LIN {X 0,Y 573.962,Z 477.903,A -85,B 0,C 180,E1 -2264.781,E2 -2264.781} C_VEL
LIN {X 0,Y 574.142,Z 465.512,A -85,B 0,C 180,E1 -2265.532,E2 -2265.532} C_VEL
LIN {X 0,Y 574.337,Z 450.828,A -85,B 0,C 180,E1 -2266.255,E2 -2266.255} C_VEL
LIN {X 0,Y 574.546,Z 436.614,A -85,B 0,C 180,E1 -2266.797,E2 -2266.797} C_VEL
LIN {X 0,Y 574.665,Z 421.538,A -85,B 0,C 180,E1 -2267.224,E2 -2267.224} C_VEL
LIN {X 0,Y 574.759,Z 406.593,A -85,B 0,C 180,E1 -2267.503,E2 -2267.503} C_VEL
LIN {X 0,Y 575.2,Z 251.055,A -85,B 0,C 180,E1 -2269.501,E2 -2269.501} C_VEL
LIN {X 0,Y 574.168,Z 244.937,A -85,B 0,C 180,E1 -2269.638,E2 -2269.638} C_VEL
LIN {X 0,Y 574.518,Z 217.413,A -85,B 0,C 180,E1 -2272.475,E2 -2272.475} C_VEL
LIN {X 0,Y 574.959,Z 188.463,A -85,B 0,C 180,E1 -2275.523,E2 -2275.523} C_VEL
LIN {X 0,Y 573.783,Z 183.004,A -85,B 0,C 180,E1 -2276.164,E2 -2276.164} C_VEL
LIN {X 0,Y 573.246,Z 180.78,A -85,B 0,C 180,E1 -2276.472,E2 -2276.472} C_VEL
LIN {X 0,Y 573.227,Z 180.7,A -85,B 0,C 180,E1 -2278.565,E2 -2278.565} C_VEL
LIN {X 0,Y 573.216,Z 180.692,A -85,B 0,C 180,E1 -2280.994,E2 -2280.994} C_VEL
LIN {X 0,Y 573.24,Z 180.703,A -85,B 0,C 180,E1 -2283.521,E2 -2283.521} C_VEL
LIN {X 0,Y 573.212,Z 180.701,A -85,B 0,C 180,E1 -2286.051,E2 -2286.051} C_VEL
LIN {X 0,Y 573.235,Z 180.708,A -85,B 0,C 180,E1 -2288.702,E2 -2288.702} C_VEL
LIN {X 0,Y 573.224,Z 180.702,A -85,B 0,C 180,E1 -2291.592,E2 -2291.592} C_VEL
LIN {X 0,Y 573.22,Z 180.705,A -85,B 0,C 180,E1 -2294.335,E2 -2294.335} C_VEL
LIN {X 0,Y 573.237,Z 180.699,A -85,B 0,C 180,E1 -2297.358,E2 -2297.358} C_VEL
LIN {X 0,Y 573.242,Z 180.706,A -85,B 0,C 180,E1 -2300.393,E2 -2300.393} C_VEL
LIN {X 0,Y 573.249,Z 180.7,A -85,B 0,C 180,E1 -2303.077,E2 -2303.077} C_VEL
LIN {X 0,Y 573.264,Z 180.697,A -85,B 0,C 180,E1 -2305.671,E2 -2305.671} C_VEL
LIN {X 0,Y 573.242,Z 180.702,A -85,B 0,C 180,E1 -2308.185,E2 -2308.185} C_VEL
LIN {X 0,Y 573.256,Z 180.702,A -85,B 0,C 180,E1 -2310.634,E2 -2310.634} C_VEL
LIN {X 0,Y 573.248,Z 180.695,A -85,B 0,C 180,E1 -2313.024,E2 -2313.024} C_VEL
LIN {X 0,Y 573.272,Z 180.695,A -85,B 0,C 180,E1 -2315.366,E2 -2315.366} C_VEL
LIN {X 0,Y 573.223,Z 180.707,A -85,B 0,C 180,E1 -2318.419,E2 -2318.419} C_VEL
LIN {X 0,Y 573.265,Z 180.697,A -85,B 0,C 180,E1 -2320.731,E2 -2320.731} C_VEL
LIN {X 0,Y 573.24,Z 180.703,A -85,B 0,C 180,E1 -2323.622,E2 -2323.622} C_VEL
LIN {X 0,Y 573.271,Z 180.702,A -85,B 0,C 180,E1 -2325.807,E2 -2325.807} C_VEL
LIN {X 0,Y 573.259,Z 180.697,A -85,B 0,C 180,E1 -2328.745,E2 -2328.745} C_VEL
LIN {X 0,Y 573.28,Z 180.699,A -85,B 0,C 180,E1 -2331.541,E2 -2331.541} C_VEL
LIN {X 0,Y 573.288,Z 180.694,A -85,B 0,C 180,E1 -2334.372,E2 -2334.372} C_VEL
LIN {X 0,Y 573.305,Z 180.696,A -85,B 0,C 180,E1 -2337.893,E2 -2337.893} C_VEL
LIN {X 0,Y 573.329,Z 180.688,A -85,B 0,C 180,E1 -2340.702,E2 -2340.702} C_VEL
LIN {X 0,Y 573.232,Z 180.708,A -85,B 0,C 180,E1 -2343.515,E2 -2343.515} C_VEL
LIN {X 0,Y 573.287,Z 180.701,A -85,B 0,C 180,E1 -2345.628,E2 -2345.628} C_VEL
LIN {X 0,Y 573.287,Z 180.693,A -85,B 0,C 180,E1 -2348.46,E2 -2348.46} C_VEL
LIN {X 0,Y 573.269,Z 180.705,A -85,B 0,C 180,E1 -2351.312,E2 -2351.312} C_VEL
LIN {X 0,Y 573.271,Z 180.696,A -85,B 0,C 180,E1 -2354.193,E2 -2354.193} C_VEL
LIN {X 0,Y 573.256,Z 180.704,A -85,B 0,C 180,E1 -2357.112,E2 -2357.112} C_VEL
LIN {X 0,Y 573.25,Z 180.697,A -85,B 0,C 180,E1 -2360.077,E2 -2360.077} C_VEL
LIN {X 0,Y 573.232,Z 180.709,A -85,B 0,C 180,E1 -2363.1,E2 -2363.1} C_VEL
LIN {X 0,Y 573.248,Z 180.699,A -85,B 0,C 180,E1 -2364.391,E2 -2364.391} C_VEL
LIN {X 0,Y 572.622,Z 180.785,A -85,B 0,C 180,E1 -2364.977,E2 -2364.977} C_VEL
LIN {X 0,Y 569.78,Z 181.138,A -85,B 0,C 180,E1 -2365.928,E2 -2365.928} C_VEL
LIN {X 0,Y 567.347,Z 181.439,A -85,B 0,C 180,E1 -2366.694,E2 -2366.694} C_VEL
LIN {X 0,Y 566.291,Z 181.568,A -85,B 0,C 180,E1 -2367.285,E2 -2367.285} C_VEL
LIN {X 0,Y 566.201,Z 181.576,A -85,B 0,C 180,E1 -2367.485,E2 -2367.485} C_VEL
LIN {X 0,Y 566.2,Z 181.575,A -85,B 0,C 180,E1 -2369.769,E2 -2369.769} C_VEL
LIN {X 0,Y 566.201,Z 181.58,A -85,B 0,C 180,E1 -2372.43,E2 -2372.43} C_VEL
LIN {X 0,Y 566.213,Z 181.58,A -85,B 0,C 180,E1 -2374.995,E2 -2374.995} C_VEL
LIN {X 0,Y 566.196,Z 181.578,A -85,B 0,C 180,E1 -2377.461,E2 -2377.461} C_VEL
LIN {X 0,Y 566.206,Z 181.576,A -85,B 0,C 180,E1 -2380.199,E2 -2380.199} C_VEL
LIN {X 0,Y 566.199,Z 181.578,A -85,B 0,C 180,E1 -2383.055,E2 -2383.055} C_VEL
LIN {X 0,Y 566.198,Z 181.58,A -85,B 0,C 180,E1 -2386.049,E2 -2386.049} C_VEL
LIN {X 0,Y 566.182,Z 181.583,A -85,B 0,C 180,E1 -2388.861,E2 -2388.861} C_VEL
LIN {X 0,Y 566.183,Z 181.579,A -85,B 0,C 180,E1 -2391.637,E2 -2391.637} C_VEL
LIN {X 0,Y 566.192,Z 181.586,A -85,B 0,C 180,E1 -2394.31,E2 -2394.31} C_VEL
LIN {X 0,Y 566.221,Z 181.573,A -85,B 0,C 180,E1 -2396.898,E2 -2396.898} C_VEL
LIN {X 0,Y 566.18,Z 181.58,A -85,B 0,C 180,E1 -2399.407,E2 -2399.407} C_VEL
LIN {X 0,Y 566.189,Z 181.586,A -85,B 0,C 180,E1 -2401.856,E2 -2401.856} C_VEL
LIN {X 0,Y 566.246,Z 181.778,A -85,B 0,C 180,E1 -2404.742,E2 -2404.742} C_VEL
LIN {X 0,Y 567.586,Z 188.138,A -85,B 0,C 180,E1 -2405.688,E2 -2405.688} C_VEL
LIN {X 0,Y 567.264,Z 206.844,A -85,B 0,C 180,E1 -2408.181,E2 -2408.181} C_VEL
LIN {X 0,Y 566.942,Z 228.424,A -85,B 0,C 180,E1 -2411.01,E2 -2411.01} C_VEL
LIN {X 0,Y 566.745,Z 244.508,A -85,B 0,C 180,E1 -2413.048,E2 -2413.048} C_VEL
LIN {X 0,Y 567.822,Z 250.993,A -85,B 0,C 180,E1 -2413.189,E2 -2413.189} C_VEL
LIN {X 0,Y 567.418,Z 382.93,A -85,B 0,C 180,E1 -2414.901,E2 -2414.901} C_VEL
LIN {X 0,Y 567.322,Z 397.304,A -85,B 0,C 180,E1 -2415.239,E2 -2415.239} C_VEL
LIN {X 0,Y 567.132,Z 411.854,A -85,B 0,C 180,E1 -2415.742,E2 -2415.742} C_VEL
LIN {X 0,Y 566.944,Z 425.536,A -85,B 0,C 180,E1 -2416.377,E2 -2416.377} C_VEL
LIN {X 0,Y 566.745,Z 437.822,A -85,B 0,C 180,E1 -2417.102,E2 -2417.102} C_VEL
LIN {X 0,Y 566.56,Z 450.215,A -85,B 0,C 180,E1 -2418.008,E2 -2418.008} C_VEL
LIN {X 0,Y 566.435,Z 461.051,A -85,B 0,C 180,E1 -2418.979,E2 -2418.979} C_VEL
LIN {X 0,Y 566.215,Z 470.48,A -85,B 0,C 180,E1 -2419.993,E2 -2419.993} C_VEL
LIN {X 0,Y 566.133,Z 478.863,A -85,B 0,C 180,E1 -2421.073,E2 -2421.073} C_VEL
LIN {X 0,Y 566.047,Z 486.874,A -85,B 0,C 180,E1 -2422.33,E2 -2422.33} C_VEL
LIN {X 0,Y 565.945,Z 493.325,A -85,B 0,C 180,E1 -2423.583,E2 -2423.583} C_VEL
LIN {X 0,Y 565.928,Z 497.799,A -85,B 0,C 180,E1 -2424.656,E2 -2424.656} C_VEL
LIN {X 0,Y 565.957,Z 501.312,A -85,B 0,C 180,E1 -2425.727,E2 -2425.727} C_VEL
LIN {X 0,Y 565.875,Z 504.745,A -85,B 0,C 180,E1 -2427.152,E2 -2427.152} C_VEL
LIN {X 0,Y 565.844,Z 506.786,A -85,B 0,C 180,E1 -2428.576,E2 -2428.576} C_VEL
LIN {X 0,Y 565.838,Z 507.496,A -85,B 0,C 180,E1 -2430,E2 -2430} C_VEL
LIN {X 0,Y 565.841,Z 506.882,A -85,B 0,C 180,E1 -2431.423,E2 -2431.423} C_VEL
LIN {X 0,Y 565.873,Z 504.926,A -85,B 0,C 180,E1 -2432.847,E2 -2432.847} C_VEL
LIN {X 0,Y 565.958,Z 501.581,A -85,B 0,C 180,E1 -2434.273,E2 -2434.273} C_VEL
LIN {X 0,Y 565.983,Z 496.748,A -85,B 0,C 180,E1 -2435.701,E2 -2435.701} C_VEL
LIN {X 0,Y 565.98,Z 490.283,A -85,B 0,C 180,E1 -2437.133,E2 -2437.133} C_VEL
LIN {X 0,Y 566.093,Z 483.082,A -85,B 0,C 180,E1 -2438.388,E2 -2438.388} C_VEL
LIN {X 0,Y 566.172,Z 475.542,A -85,B 0,C 180,E1 -2439.466,E2 -2439.466} C_VEL
LIN {X 0,Y 566.29,Z 466.488,A -85,B 0,C 180,E1 -2440.547,E2 -2440.547} C_VEL
LIN {X 0,Y 566.47,Z 455.522,A -85,B 0,C 180,E1 -2441.631,E2 -2441.631} C_VEL
LIN {X 0,Y 566.642,Z 444.356,A -85,B 0,C 180,E1 -2442.535,E2 -2442.535} C_VEL
LIN {X 0,Y 566.843,Z 432.011,A -85,B 0,C 180,E1 -2443.351,E2 -2443.351} C_VEL
LIN {X 0,Y 567.065,Z 420.127,A -85,B 0,C 180,E1 -2443.985,E2 -2443.985} C_VEL
LIN {X 0,Y 567.232,Z 407.918,A -85,B 0,C 180,E1 -2444.503,E2 -2444.503} C_VEL
LIN {X 0,Y 567.343,Z 393.992,A -85,B 0,C 180,E1 -2444.943,E2 -2444.943} C_VEL
LIN {X 0,Y 567.428,Z 380.103,A -85,B 0,C 180,E1 -2445.236,E2 -2445.236} C_VEL
LIN {X 0,Y 567.751,Z 250.574,A -85,B 0,C 180,E1 -2446.908,E2 -2446.908} C_VEL
LIN {X 0,Y 566.728,Z 244.432,A -85,B 0,C 180,E1 -2447.047,E2 -2447.047} C_VEL
LIN {X 0,Y 566.979,Z 224.441,A -85,B 0,C 180,E1 -2449.599,E2 -2449.599} C_VEL
LIN {X 0,Y 567.381,Z 201.774,A -85,B 0,C 180,E1 -2452.58,E2 -2452.58} C_VEL
LIN {X 0,Y 567.58,Z 188.81,A -85,B 0,C 180,E1 -2454.312,E2 -2454.312} C_VEL
LIN {X 0,Y 566.223,Z 181.721,A -85,B 0,C 180,E1 -2455.363,E2 -2455.363} C_VEL
LIN {X 0,Y 566.184,Z 181.587,A -85,B 0,C 180,E1 -2458.198,E2 -2458.198} C_VEL
LIN {X 0,Y 566.188,Z 181.579,A -85,B 0,C 180,E1 -2461.075,E2 -2461.075} C_VEL
LIN {X 0,Y 566.21,Z 181.578,A -85,B 0,C 180,E1 -2463.733,E2 -2463.733} C_VEL
LIN {X 0,Y 566.212,Z 181.575,A -85,B 0,C 180,E1 -2466.568,E2 -2466.568} C_VEL
LIN {X 0,Y 566.212,Z 181.583,A -85,B 0,C 180,E1 -2469.685,E2 -2469.685} C_VEL
LIN {X 0,Y 566.21,Z 181.577,A -85,B 0,C 180,E1 -2472.087,E2 -2472.087} C_VEL
LIN {X 0,Y 566.17,Z 181.583,A -85,B 0,C 180,E1 -2475.035,E2 -2475.035} C_VEL
LIN {X 0,Y 566.214,Z 181.576,A -85,B 0,C 180,E1 -2478.135,E2 -2478.135} C_VEL
LIN {X 0,Y 566.211,Z 181.574,A -85,B 0,C 180,E1 -2480.726,E2 -2480.726} C_VEL
LIN {X 0,Y 566.213,Z 181.577,A -85,B 0,C 180,E1 -2483.783,E2 -2483.783} C_VEL
LIN {X 0,Y 566.207,Z 181.574,A -85,B 0,C 180,E1 -2486.265,E2 -2486.265} C_VEL
LIN {X 0,Y 566.193,Z 181.583,A -85,B 0,C 180,E1 -2488.922,E2 -2488.922} C_VEL
LIN {X 0,Y 566.19,Z 181.582,A -85,B 0,C 180,E1 -2491.046,E2 -2491.046} C_VEL
LIN {X 0,Y 566.21,Z 181.579,A -85,B 0,C 180,E1 -2493.458,E2 -2493.458} C_VEL
LIN {X 0,Y 566.193,Z 181.577,A -85,B 0,C 180,E1 -2495.819,E2 -2495.819} C_VEL
LIN {X 0,Y 566.202,Z 181.586,A -85,B 0,C 180,E1 -2498.902,E2 -2498.902} C_VEL
LIN {X 0,Y 566.206,Z 181.581,A -85,B 0,C 180,E1 -2501.172,E2 -2501.172} C_VEL
LIN {X 0,Y 566.215,Z 181.575,A -85,B 0,C 180,E1 -2503.412,E2 -2503.412} C_VEL
LIN {X 0,Y 566.195,Z 181.581,A -85,B 0,C 180,E1 -2506.359,E2 -2506.359} C_VEL
LIN {X 0,Y 566.227,Z 181.581,A -85,B 0,C 180,E1 -2508.675,E2 -2508.675} C_VEL
LIN {X 0,Y 566.227,Z 181.573,A -85,B 0,C 180,E1 -2511.434,E2 -2511.434} C_VEL
LIN {X 0,Y 566.254,Z 181.575,A -85,B 0,C 180,E1 -2514.302,E2 -2514.302} C_VEL
LIN {X 0,Y 566.274,Z 181.568,A -85,B 0,C 180,E1 -2517.866,E2 -2517.866} C_VEL
LIN {X 0,Y 566.298,Z 181.567,A -85,B 0,C 180,E1 -2520.711,E2 -2520.711} C_VEL
LIN {X 0,Y 566.267,Z 181.571,A -85,B 0,C 180,E1 -2522.845,E2 -2522.845} C_VEL
LIN {X 0,Y 566.255,Z 181.57,A -85,B 0,C 180,E1 -2525.698,E2 -2525.698} C_VEL
LIN {X 0,Y 566.227,Z 181.576,A -85,B 0,C 180,E1 -2528.566,E2 -2528.566} C_VEL
LIN {X 0,Y 566.234,Z 181.573,A -85,B 0,C 180,E1 -2531.454,E2 -2531.454} C_VEL
LIN {X 0,Y 566.227,Z 181.576,A -85,B 0,C 180,E1 -2534.507,E2 -2534.507} C_VEL
LIN {X 0,Y 566.196,Z 181.578,A -85,B 0,C 180,E1 -2537.332,E2 -2537.332} C_VEL
LIN {X 0,Y 566.205,Z 181.578,A -85,B 0,C 180,E1 -2540.337,E2 -2540.337} C_VEL
LIN {X 0,Y 566.182,Z 181.582,A -85,B 0,C 180,E1 -2543.404,E2 -2543.404} C_VEL
LIN {X 0,Y 566.219,Z 181.579,A -85,B 0,C 180,E1 -2545.749,E2 -2545.749} C_VEL
LIN {X 0,Y 566.195,Z 181.579,A -85,B 0,C 180,E1 -2548.202,E2 -2548.202} C_VEL
LIN {X 0,Y 566.187,Z 181.58,A -85,B 0,C 180,E1 -2551.078,E2 -2551.078} C_VEL
LIN {X 0,Y 566.205,Z 181.583,A -85,B 0,C 180,E1 -2553.735,E2 -2553.735} C_VEL
LIN {X 0,Y 566.201,Z 181.576,A -85,B 0,C 180,E1 -2556.57,E2 -2556.57} C_VEL
LIN {X 0,Y 566.215,Z 181.58,A -85,B 0,C 180,E1 -2559.687,E2 -2559.687} C_VEL
LIN {X 0,Y 566.195,Z 181.579,A -85,B 0,C 180,E1 -2562.918,E2 -2562.918} C_VEL
LIN {X 0,Y 566.188,Z 181.578,A -85,B 0,C 180,E1 -2566.05,E2 -2566.05} C_VEL
LIN {X 0,Y 566.198,Z 181.579,A -85,B 0,C 180,E1 -2569.215,E2 -2569.215} C_VEL
LIN {X 0,Y 566.177,Z 181.582,A -85,B 0,C 180,E1 -2571.637,E2 -2571.637} C_VEL
LIN {X 0,Y 566.157,Z 181.58,A -85,B 0,C 180,E1 -2574.308,E2 -2574.308} C_VEL
LIN {X 0,Y 566.195,Z 181.586,A -85,B 0,C 180,E1 -2576.897,E2 -2576.897} C_VEL
LIN {X 0,Y 566.165,Z 181.563,A -85,B 0,C 180,E1 -2579.407,E2 -2579.407} C_VEL
LIN {X 0,Y 566.187,Z 181.583,A -85,B 0,C 180,E1 -2581.857,E2 -2581.857} C_VEL
LIN {X 0,Y 566.194,Z 181.774,A -85,B 0,C 180,E1 -2583.318,E2 -2583.318} C_VEL
LIN {X 0,Y 568.156,Z 190.164,A -85,B 0,C 180,E1 -2584.346,E2 -2584.346} C_VEL
LIN {X 0,Y 567.675,Z 217.287,A -85,B 0,C 180,E1 -2587.24,E2 -2587.24} C_VEL
LIN {X 0,Y 567.331,Z 244.836,A -85,B 0,C 180,E1 -2590.108,E2 -2590.108} C_VEL
LIN {X 0,Y 568.527,Z 252.976,A -85,B 0,C 180,E1 -2590.286,E2 -2590.286} C_VEL
LIN {X 0,Y 568.009,Z 411.919,A -85,B 0,C 180,E1 -2592.364,E2 -2592.364} C_VEL
LIN {X 0,Y 567.848,Z 427.721,A -85,B 0,C 180,E1 -2592.721,E2 -2592.721} C_VEL
LIN {X 0,Y 567.617,Z 443.049,A -85,B 0,C 180,E1 -2593.224,E2 -2593.224} C_VEL
LIN {X 0,Y 567.429,Z 456.787,A -85,B 0,C 180,E1 -2593.819,E2 -2593.819} C_VEL
LIN {X 0,Y 567.173,Z 470.257,A -85,B 0,C 180,E1 -2594.55,E2 -2594.55} C_VEL
LIN {X 0,Y 566.931,Z 482.529,A -85,B 0,C 180,E1 -2595.359,E2 -2595.359} C_VEL
LIN {X 0,Y 566.672,Z 495.297,A -85,B 0,C 180,E1 -2596.371,E2 -2596.371} C_VEL
LIN {X 0,Y 566.491,Z 506.754,A -85,B 0,C 180,E1 -2597.461,E2 -2597.461} C_VEL
LIN {X 0,Y 566.268,Z 517.314,A -85,B 0,C 180,E1 -2598.659,E2 -2598.659} C_VEL
LIN {X 0,Y 566.208,Z 525.859,A -85,B 0,C 180,E1 -2599.813,E2 -2599.813} C_VEL
LIN {X 0,Y 566.057,Z 533.737,A -85,B 0,C 180,E1 -2601.072,E2 -2601.072} C_VEL
LIN {X 0,Y 565.997,Z 541.091,A -85,B 0,C 180,E1 -2602.509,E2 -2602.509} C_VEL
LIN {X 0,Y 565.959,Z 546.924,A -85,B 0,C 180,E1 -2603.941,E2 -2603.941} C_VEL
LIN {X 0,Y 565.866,Z 550.387,A -85,B 0,C 180,E1 -2605.013,E2 -2605.013} C_VEL
LIN {X 0,Y 565.909,Z 553.89,A -85,B 0,C 180,E1 -2606.44,E2 -2606.44} C_VEL
LIN {X 0,Y 565.839,Z 556.192,A -85,B 0,C 180,E1 -2607.865,E2 -2607.865} C_VEL
LIN {X 0,Y 565.839,Z 557.349,A -85,B 0,C 180,E1 -2609.289,E2 -2609.289} C_VEL
LIN {X 0,Y 565.839,Z 557.348,A -85,B 0,C 180,E1 -2610.712,E2 -2610.712} C_VEL
LIN {X 0,Y 565.839,Z 556.189,A -85,B 0,C 180,E1 -2612.136,E2 -2612.136} C_VEL
LIN {X 0,Y 565.909,Z 553.886,A -85,B 0,C 180,E1 -2613.56,E2 -2613.56} C_VEL
LIN {X 0,Y 565.867,Z 550.385,A -85,B 0,C 180,E1 -2614.988,E2 -2614.988} C_VEL
LIN {X 0,Y 565.943,Z 545.608,A -85,B 0,C 180,E1 -2616.417,E2 -2616.417} C_VEL
LIN {X 0,Y 566.014,Z 539.421,A -85,B 0,C 180,E1 -2617.85,E2 -2617.85} C_VEL
LIN {X 0,Y 566.071,Z 531.646,A -85,B 0,C 180,E1 -2619.288,E2 -2619.288} C_VEL
LIN {X 0,Y 566.24,Z 523.367,A -85,B 0,C 180,E1 -2620.549,E2 -2620.549} C_VEL
LIN {X 0,Y 566.367,Z 513.39,A -85,B 0,C 180,E1 -2621.815,E2 -2621.815} C_VEL
LIN {X 0,Y 566.586,Z 503.186,A -85,B 0,C 180,E1 -2622.901,E2 -2622.901} C_VEL
LIN {X 0,Y 566.8,Z 491.018,A -85,B 0,C 180,E1 -2623.992,E2 -2623.992} C_VEL
LIN {X 0,Y 567.04,Z 478.337,A -85,B 0,C 180,E1 -2624.936,E2 -2624.936} C_VEL
LIN {X 0,Y 567.278,Z 465.509,A -85,B 0,C 180,E1 -2625.724,E2 -2625.724} C_VEL
LIN {X 0,Y 567.499,Z 450.825,A -85,B 0,C 180,E1 -2626.457,E2 -2626.457} C_VEL
LIN {X 0,Y 567.752,Z 436.613,A -85,B 0,C 180,E1 -2627.004,E2 -2627.004} C_VEL
LIN {X 0,Y 567.871,Z 422.181,A -85,B 0,C 180,E1 -2627.421,E2 -2627.421} C_VEL
LIN {X 0,Y 568.016,Z 406.62,A -85,B 0,C 180,E1 -2627.718,E2 -2627.718} C_VEL
LIN {X 0,Y 568.416,Z 251.099,A -85,B 0,C 180,E1 -2629.742,E2 -2629.742} C_VEL
LIN {X 0,Y 567.317,Z 244.916,A -85,B 0,C 180,E1 -2629.887,E2 -2629.887} C_VEL
LIN {X 0,Y 567.677,Z 217.282,A -85,B 0,C 180,E1 -2632.761,E2 -2632.761} C_VEL
LIN {X 0,Y 568.183,Z 190.159,A -85,B 0,C 180,E1 -2635.653,E2 -2635.653} C_VEL
LIN {X 0,Y 566.204,Z 181.721,A -85,B 0,C 180,E1 -2636.694,E2 -2636.694} C_VEL
LIN {X 0,Y 566.173,Z 181.563,A -85,B 0,C 180,E1 -2638.954,E2 -2638.954} C_VEL
LIN {X 0,Y 566.187,Z 181.577,A -85,B 0,C 180,E1 -2641.422,E2 -2641.422} C_VEL
LIN {X 0,Y 566.195,Z 181.578,A -85,B 0,C 180,E1 -2643.957,E2 -2643.957} C_VEL
LIN {X 0,Y 566.197,Z 181.579,A -85,B 0,C 180,E1 -2646.57,E2 -2646.57} C_VEL
LIN {X 0,Y 566.211,Z 181.568,A -85,B 0,C 180,E1 -2649.685,E2 -2649.685} C_VEL
LIN {X 0,Y 566.199,Z 181.584,A -85,B 0,C 180,E1 -2652.917,E2 -2652.917} C_VEL
LIN {X 0,Y 566.191,Z 181.579,A -85,B 0,C 180,E1 -2656.049,E2 -2656.049} C_VEL
LIN {X 0,Y 566.201,Z 181.578,A -85,B 0,C 180,E1 -2659.214,E2 -2659.214} C_VEL
LIN {X 0,Y 566.182,Z 181.578,A -85,B 0,C 180,E1 -2661.637,E2 -2661.637} C_VEL
LIN {X 0,Y 566.161,Z 181.588,A -85,B 0,C 180,E1 -2664.308,E2 -2664.308} C_VEL
LIN {X 0,Y 566.217,Z 181.574,A -85,B 0,C 180,E1 -2666.898,E2 -2666.898} C_VEL
LIN {X 0,Y 566.174,Z 181.579,A -85,B 0,C 180,E1 -2669.407,E2 -2669.407} C_VEL
LIN {X 0,Y 566.208,Z 181.578,A -85,B 0,C 180,E1 -2671.857,E2 -2671.857} C_VEL
LIN {X 0,Y 566.213,Z 181.58,A -85,B 0,C 180,E1 -2674.251,E2 -2674.251} C_VEL
LIN {X 0,Y 566.169,Z 181.583,A -85,B 0,C 180,E1 -2676.718,E2 -2676.718} C_VEL
LIN {X 0,Y 566.208,Z 181.578,A -85,B 0,C 180,E1 -2679.663,E2 -2679.663} C_VEL
LIN {X 0,Y 566.199,Z 181.578,A -85,B 0,C 180,E1 -2682.668,E2 -2682.668} C_VEL
LIN {X 0,Y 566.231,Z 181.577,A -85,B 0,C 180,E1 -2685.627,E2 -2685.627} C_VEL
LIN {X 0,Y 566.231,Z 181.573,A -85,B 0,C 180,E1 -2688.675,E2 -2688.675} C_VEL
LIN {X 0,Y 566.224,Z 181.576,A -85,B 0,C 180,E1 -2691.434,E2 -2691.434} C_VEL
LIN {X 0,Y 566.256,Z 181.57,A -85,B 0,C 180,E1 -2694.302,E2 -2694.302} C_VEL
LIN {X 0,Y 566.276,Z 181.572,A -85,B 0,C 180,E1 -2697.866,E2 -2697.866} C_VEL
LIN {X 0,Y 566.299,Z 181.564,A -85,B 0,C 180,E1 -2700.711,E2 -2700.711} C_VEL
LIN {X 0,Y 566.271,Z 181.567,A -85,B 0,C 180,E1 -2702.846,E2 -2702.846} C_VEL
LIN {X 0,Y 566.255,Z 181.576,A -85,B 0,C 180,E1 -2705.698,E2 -2705.698} C_VEL
LIN {X 0,Y 566.23,Z 181.572,A -85,B 0,C 180,E1 -2708.566,E2 -2708.566} C_VEL
LIN {X 0,Y 566.239,Z 181.579,A -85,B 0,C 180,E1 -2711.455,E2 -2711.455} C_VEL
LIN {X 0,Y 566.232,Z 181.573,A -85,B 0,C 180,E1 -2714.507,E2 -2714.507} C_VEL
LIN {X 0,Y 566.198,Z 181.585,A -85,B 0,C 180,E1 -2717.332,E2 -2717.332} C_VEL
LIN {X 0,Y 566.211,Z 181.574,A -85,B 0,C 180,E1 -2720.337,E2 -2720.337} C_VEL
LIN {X 0,Y 566.171,Z 181.586,A -85,B 0,C 180,E1 -2723.282,E2 -2723.282} C_VEL
LIN {X 0,Y 566.211,Z 181.576,A -85,B 0,C 180,E1 -2725.749,E2 -2725.749} C_VEL
LIN {X 0,Y 566.201,Z 181.576,A -85,B 0,C 180,E1 -2727.485,E2 -2727.485} C_VEL
LIN {X 0,Y 565.521,Z 181.66,A -85,B 0,C 180,E1 -2728.079,E2 -2728.079} C_VEL
LIN {X 0,Y 562.655,Z 182.022,A -85,B 0,C 180,E1 -2729.043,E2 -2729.043} C_VEL
LIN {X 0,Y 560.246,Z 182.319,A -85,B 0,C 180,E1 -2729.818,E2 -2729.818} C_VEL
LIN {X 0,Y 559.218,Z 182.447,A -85,B 0,C 180,E1 -2730.417,E2 -2730.417} C_VEL
LIN {X 0,Y 559.138,Z 182.458,A -85,B 0,C 180,E1 -2730.62,E2 -2730.62} C_VEL
LIN {X 0,Y 559.162,Z 182.452,A -85,B 0,C 180,E1 -2733.575,E2 -2733.575} C_VEL
LIN {X 0,Y 559.168,Z 182.456,A -85,B 0,C 180,E1 -2736.449,E2 -2736.449} C_VEL
LIN {X 0,Y 559.174,Z 182.454,A -85,B 0,C 180,E1 -2738.934,E2 -2738.934} C_VEL
LIN {X 0,Y 559.162,Z 182.454,A -85,B 0,C 180,E1 -2741.771,E2 -2741.771} C_VEL
LIN {X 0,Y 559.135,Z 182.464,A -85,B 0,C 180,E1 -2744.74,E2 -2744.74} C_VEL
LIN {X 0,Y 559.162,Z 182.452,A -85,B 0,C 180,E1 -2747.257,E2 -2747.257} C_VEL
LIN {X 0,Y 559.179,Z 182.457,A -85,B 0,C 180,E1 -2750.135,E2 -2750.135} C_VEL
LIN {X 0,Y 559.143,Z 182.457,A -85,B 0,C 180,E1 -2752.892,E2 -2752.892} C_VEL
LIN {X 0,Y 559.167,Z 182.459,A -85,B 0,C 180,E1 -2756.051,E2 -2756.051} C_VEL
LIN {X 0,Y 559.155,Z 182.455,A -85,B 0,C 180,E1 -2758.981,E2 -2758.981} C_VEL
LIN {X 0,Y 559.136,Z 182.462,A -85,B 0,C 180,E1 -2761.626,E2 -2761.626} C_VEL
LIN {X 0,Y 559.196,Z 182.624,A -85,B 0,C 180,E1 -2764.504,E2 -2764.504} C_VEL
LIN {X 0,Y 560.728,Z 189.676,A -85,B 0,C 180,E1 -2765.568,E2 -2765.568} C_VEL
LIN {X 0,Y 560.437,Z 206.957,A -85,B 0,C 180,E1 -2767.901,E2 -2767.901} C_VEL
LIN {X 0,Y 560.036,Z 228.72,A -85,B 0,C 180,E1 -2770.789,E2 -2770.789} C_VEL
LIN {X 0,Y 559.818,Z 244.356,A -85,B 0,C 180,E1 -2772.814,E2 -2772.814} C_VEL
LIN {X 0,Y 560.625,Z 249.285,A -85,B 0,C 180,E1 -2772.94,E2 -2772.94} C_VEL
LIN {X 0,Y 561.01,Z 252.625,A -85,B 0,C 180,E1 -2772.998,E2 -2772.998} C_VEL
LIN {X 0,Y 560.583,Z 382.959,A -85,B 0,C 180,E1 -2774.712,E2 -2774.712} C_VEL
LIN {X 0,Y 560.457,Z 397.502,A -85,B 0,C 180,E1 -2775.06,E2 -2775.06} C_VEL
LIN {X 0,Y 560.238,Z 411.867,A -85,B 0,C 180,E1 -2775.562,E2 -2775.562} C_VEL
LIN {X 0,Y 560.036,Z 425.545,A -85,B 0,C 180,E1 -2776.206,E2 -2776.206} C_VEL
LIN {X 0,Y 559.813,Z 437.834,A -85,B 0,C 180,E1 -2776.94,E2 -2776.94} C_VEL
LIN {X 0,Y 559.57,Z 450.222,A -85,B 0,C 180,E1 -2777.856,E2 -2777.856} C_VEL
LIN {X 0,Y 559.417,Z 461.297,A -85,B 0,C 180,E1 -2778.864,E2 -2778.864} C_VEL
LIN {X 0,Y 559.201,Z 470.486,A -85,B 0,C 180,E1 -2779.866,E2 -2779.866} C_VEL
LIN {X 0,Y 559.071,Z 478.867,A -85,B 0,C 180,E1 -2780.959,E2 -2780.959} C_VEL
LIN {X 0,Y 558.974,Z 486.877,A -85,B 0,C 180,E1 -2782.232,E2 -2782.232} C_VEL
LIN {X 0,Y 558.873,Z 493.327,A -85,B 0,C 180,E1 -2783.501,E2 -2783.501} C_VEL
LIN {X 0,Y 558.859,Z 497.801,A -85,B 0,C 180,E1 -2784.588,E2 -2784.588} C_VEL
LIN {X 0,Y 558.866,Z 501.314,A -85,B 0,C 180,E1 -2785.673,E2 -2785.673} C_VEL
LIN {X 0,Y 558.796,Z 504.747,A -85,B 0,C 180,E1 -2787.116,E2 -2787.116} C_VEL
LIN {X 0,Y 558.744,Z 506.788,A -85,B 0,C 180,E1 -2788.558,E2 -2788.558} C_VEL
LIN {X 0,Y 558.739,Z 507.496,A -85,B 0,C 180,E1 -2790,E2 -2790} C_VEL
LIN {X 0,Y 558.741,Z 506.882,A -85,B 0,C 180,E1 -2791.441,E2 -2791.441} C_VEL
LIN {X 0,Y 558.794,Z 504.926,A -85,B 0,C 180,E1 -2792.883,E2 -2792.883} C_VEL
LIN {X 0,Y 558.867,Z 501.58,A -85,B 0,C 180,E1 -2794.327,E2 -2794.327} C_VEL
LIN {X 0,Y 558.912,Z 496.746,A -85,B 0,C 180,E1 -2795.773,E2 -2795.773} C_VEL
LIN {X 0,Y 558.907,Z 490.281,A -85,B 0,C 180,E1 -2797.223,E2 -2797.223} C_VEL
LIN {X 0,Y 559.028,Z 483.079,A -85,B 0,C 180,E1 -2798.494,E2 -2798.494} C_VEL
LIN {X 0,Y 559.124,Z 475.538,A -85,B 0,C 180,E1 -2799.587,E2 -2799.587} C_VEL
LIN {X 0,Y 559.287,Z 466.482,A -85,B 0,C 180,E1 -2800.681,E2 -2800.681} C_VEL
LIN {X 0,Y 559.486,Z 457.47,A -85,B 0,C 180,E1 -2801.594,E2 -2801.594} C_VEL
LIN {X 0,Y 559.629,Z 446.716,A -85,B 0,C 180,E1 -2802.511,E2 -2802.511} C_VEL
LIN {X 0,Y 559.842,Z 434.951,A -85,B 0,C 180,E1 -2803.336,E2 -2803.336} C_VEL
LIN {X 0,Y 560.107,Z 421.97,A -85,B 0,C 180,E1 -2804.07,E2 -2804.07} C_VEL
LIN {X 0,Y 560.35,Z 408.189,A -85,B 0,C 180,E1 -2804.675,E2 -2804.675} C_VEL
LIN {X 0,Y 560.493,Z 393.869,A -85,B 0,C 180,E1 -2805.133,E2 -2805.133} C_VEL
LIN {X 0,Y 560.572,Z 380.065,A -85,B 0,C 180,E1 -2805.427,E2 -2805.427} C_VEL
LIN {X 0,Y 560.988,Z 251.597,A -85,B 0,C 180,E1 -2807.106,E2 -2807.106} C_VEL
LIN {X 0,Y 559.795,Z 244.499,A -85,B 0,C 180,E1 -2807.267,E2 -2807.267} C_VEL
LIN {X 0,Y 560.09,Z 225.206,A -85,B 0,C 180,E1 -2809.763,E2 -2809.763} C_VEL
LIN {X 0,Y 560.544,Z 201.88,A -85,B 0,C 180,E1 -2812.871,E2 -2812.871} C_VEL
LIN {X 0,Y 560.738,Z 190.339,A -85,B 0,C 180,E1 -2814.431,E2 -2814.431} C_VEL
LIN {X 0,Y 559.165,Z 182.548,A -85,B 0,C 180,E1 -2815.614,E2 -2815.614} C_VEL
LIN {X 0,Y 559.13,Z 182.462,A -85,B 0,C 180,E1 -2818.531,E2 -2818.531} C_VEL
LIN {X 0,Y 559.144,Z 182.458,A -85,B 0,C 180,E1 -2821.272,E2 -2821.272} C_VEL
LIN {X 0,Y 559.164,Z 182.458,A -85,B 0,C 180,E1 -2823.948,E2 -2823.948} C_VEL
LIN {X 0,Y 559.144,Z 182.456,A -85,B 0,C 180,E1 -2827.107,E2 -2827.107} C_VEL
LIN {X 0,Y 559.158,Z 182.46,A -85,B 0,C 180,E1 -2829.941,E2 -2829.941} C_VEL
LIN {X 0,Y 559.158,Z 182.453,A -85,B 0,C 180,E1 -2832.743,E2 -2832.743} C_VEL
LIN {X 0,Y 559.149,Z 182.46,A -85,B 0,C 180,E1 -2835.76,E2 -2835.76} C_VEL
LIN {X 0,Y 559.187,Z 182.451,A -85,B 0,C 180,E1 -2838.232,E2 -2838.232} C_VEL
LIN {X 0,Y 559.17,Z 182.456,A -85,B 0,C 180,E1 -2841.191,E2 -2841.191} C_VEL
LIN {X 0,Y 559.168,Z 182.454,A -85,B 0,C 180,E1 -2843.791,E2 -2843.791} C_VEL
LIN {X 0,Y 559.16,Z 182.452,A -85,B 0,C 180,E1 -2846.425,E2 -2846.425} C_VEL
LIN {X 0,Y 559.157,Z 182.46,A -85,B 0,C 180,E1 -2848.981,E2 -2848.981} C_VEL
LIN {X 0,Y 559.165,Z 182.452,A -85,B 0,C 180,E1 -2851.618,E2 -2851.618} C_VEL
LIN {X 0,Y 559.175,Z 182.452,A -85,B 0,C 180,E1 -2853.902,E2 -2853.902} C_VEL
LIN {X 0,Y 559.15,Z 182.457,A -85,B 0,C 180,E1 -2856.567,E2 -2856.567} C_VEL
LIN {X 0,Y 559.174,Z 182.453,A -85,B 0,C 180,E1 -2859.395,E2 -2859.395} C_VEL
LIN {X 0,Y 559.148,Z 182.455,A -85,B 0,C 180,E1 -2861.686,E2 -2861.686} C_VEL
LIN {X 0,Y 559.165,Z 182.452,A -85,B 0,C 180,E1 -2863.948,E2 -2863.948} C_VEL
LIN {X 0,Y 559.169,Z 182.454,A -85,B 0,C 180,E1 -2866.184,E2 -2866.184} C_VEL
LIN {X 0,Y 559.188,Z 182.453,A -85,B 0,C 180,E1 -2869.133,E2 -2869.133} C_VEL
LIN {X 0,Y 559.2,Z 182.45,A -85,B 0,C 180,E1 -2872.053,E2 -2872.053} C_VEL
LIN {X 0,Y 559.25,Z 182.445,A -85,B 0,C 180,E1 -2874.953,E2 -2874.953} C_VEL
LIN {X 0,Y 559.245,Z 182.443,A -85,B 0,C 180,E1 -2877.839,E2 -2877.839} C_VEL
LIN {X 0,Y 559.268,Z 182.443,A -85,B 0,C 180,E1 -2880.72,E2 -2880.72} C_VEL
LIN {X 0,Y 559.233,Z 182.446,A -85,B 0,C 180,E1 -2882.881,E2 -2882.881} C_VEL
LIN {X 0,Y 559.225,Z 182.446,A -85,B 0,C 180,E1 -2885.77,E2 -2885.77} C_VEL
LIN {X 0,Y 559.185,Z 182.452,A -85,B 0,C 180,E1 -2888.674,E2 -2888.674} C_VEL
LIN {X 0,Y 559.197,Z 182.451,A -85,B 0,C 180,E1 -2891.6,E2 -2891.6} C_VEL
LIN {X 0,Y 559.192,Z 182.451,A -85,B 0,C 180,E1 -2894.596,E2 -2894.596} C_VEL
LIN {X 0,Y 559.156,Z 182.457,A -85,B 0,C 180,E1 -2897.557,E2 -2897.557} C_VEL
LIN {X 0,Y 559.164,Z 182.461,A -85,B 0,C 180,E1 -2899.838,E2 -2899.838} C_VEL
LIN {X 0,Y 559.133,Z 182.462,A -85,B 0,C 180,E1 -2902.153,E2 -2902.153} C_VEL
LIN {X 0,Y 559.173,Z 182.452,A -85,B 0,C 180,E1 -2905.188,E2 -2905.188} C_VEL
LIN {X 0,Y 559.177,Z 182.456,A -85,B 0,C 180,E1 -2907.712,E2 -2907.712} C_VEL
LIN {X 0,Y 559.145,Z 182.457,A -85,B 0,C 180,E1 -2910.183,E2 -2910.183} C_VEL
LIN {X 0,Y 559.168,Z 182.448,A -85,B 0,C 180,E1 -2912.714,E2 -2912.714} C_VEL
LIN {X 0,Y 559.143,Z 182.462,A -85,B 0,C 180,E1 -2915.323,E2 -2915.323} C_VEL
LIN {X 0,Y 559.127,Z 182.458,A -85,B 0,C 180,E1 -2918.018,E2 -2918.018} C_VEL
LIN {X 0,Y 559.149,Z 182.457,A -85,B 0,C 180,E1 -2920.813,E2 -2920.813} C_VEL
LIN {X 0,Y 559.132,Z 182.461,A -85,B 0,C 180,E1 -2923.735,E2 -2923.735} C_VEL
LIN {X 0,Y 559.139,Z 182.459,A -85,B 0,C 180,E1 -2926.804,E2 -2926.804} C_VEL
LIN {X 0,Y 559.15,Z 182.456,A -85,B 0,C 180,E1 -2929.188,E2 -2929.188} C_VEL
LIN {X 0,Y 559.126,Z 182.459,A -85,B 0,C 180,E1 -2931.983,E2 -2931.983} C_VEL
LIN {X 0,Y 559.126,Z 182.459,A -85,B 0,C 180,E1 -2934.788,E2 -2934.788} C_VEL
LIN {X 0,Y 559.148,Z 182.457,A -85,B 0,C 180,E1 -2937.366,E2 -2937.366} C_VEL
LIN {X 0,Y 559.117,Z 182.435,A -85,B 0,C 180,E1 -2940.148,E2 -2940.148} C_VEL
LIN {X 0,Y 559.149,Z 182.58,A -85,B 0,C 180,E1 -2943.047,E2 -2943.047} C_VEL
LIN {X 0,Y 561.284,Z 191.115,A -85,B 0,C 180,E1 -2944.126,E2 -2944.126} C_VEL
LIN {X 0,Y 561.066,Z 208.019,A -85,B 0,C 180,E1 -2945.965,E2 -2945.965} C_VEL
LIN {X 0,Y 560.595,Z 233.443,A -85,B 0,C 180,E1 -2948.681,E2 -2948.681} C_VEL
LIN {X 0,Y 560.468,Z 244.975,A -85,B 0,C 180,E1 -2949.87,E2 -2949.87} C_VEL
LIN {X 0,Y 561.838,Z 253.562,A -85,B 0,C 180,E1 -2950.052,E2 -2950.052} C_VEL
LIN {X 0,Y 561.247,Z 411.715,A -85,B 0,C 180,E1 -2952.141,E2 -2952.141} C_VEL
LIN {X 0,Y 561.052,Z 427.719,A -85,B 0,C 180,E1 -2952.505,E2 -2952.505} C_VEL
LIN {X 0,Y 560.826,Z 443.047,A -85,B 0,C 180,E1 -2953.014,E2 -2953.014} C_VEL
LIN {X 0,Y 560.589,Z 456.79,A -85,B 0,C 180,E1 -2953.616,E2 -2953.616} C_VEL
LIN {X 0,Y 560.302,Z 470.26,A -85,B 0,C 180,E1 -2954.355,E2 -2954.355} C_VEL
LIN {X 0,Y 559.997,Z 483.31,A -85,B 0,C 180,E1 -2955.231,E2 -2955.231} C_VEL
LIN {X 0,Y 559.722,Z 495.298,A -85,B 0,C 180,E1 -2956.198,E2 -2956.198} C_VEL
LIN {X 0,Y 559.515,Z 506.754,A -85,B 0,C 180,E1 -2957.302,E2 -2957.302} C_VEL
LIN {X 0,Y 559.303,Z 516.392,A -85,B 0,C 180,E1 -2958.402,E2 -2958.402} C_VEL
LIN {X 0,Y 559.168,Z 525.858,A -85,B 0,C 180,E1 -2959.683,E2 -2959.683} C_VEL
LIN {X 0,Y 559.002,Z 533.737,A -85,B 0,C 180,E1 -2960.959,E2 -2960.959} C_VEL
LIN {X 0,Y 558.92,Z 541.092,A -85,B 0,C 180,E1 -2962.413,E2 -2962.413} C_VEL
LIN {X 0,Y 558.859,Z 546.923,A -85,B 0,C 180,E1 -2963.864,E2 -2963.864} C_VEL
LIN {X 0,Y 558.787,Z 550.387,A -85,B 0,C 180,E1 -2964.949,E2 -2964.949} C_VEL
LIN {X 0,Y 558.818,Z 553.889,A -85,B 0,C 180,E1 -2966.395,E2 -2966.395} C_VEL
LIN {X 0,Y 558.745,Z 556.191,A -85,B 0,C 180,E1 -2967.838,E2 -2967.838} C_VEL
LIN {X 0,Y 558.739,Z 557.348,A -85,B 0,C 180,E1 -2969.28,E2 -2969.28} C_VEL
LIN {X 0,Y 558.739,Z 557.348,A -85,B 0,C 180,E1 -2970.721,E2 -2970.721} C_VEL
LIN {X 0,Y 558.745,Z 556.188,A -85,B 0,C 180,E1 -2972.163,E2 -2972.163} C_VEL
LIN {X 0,Y 558.818,Z 553.885,A -85,B 0,C 180,E1 -2973.606,E2 -2973.606} C_VEL
LIN {X 0,Y 558.787,Z 550.386,A -85,B 0,C 180,E1 -2975.051,E2 -2975.051} C_VEL
LIN {X 0,Y 558.871,Z 545.608,A -85,B 0,C 180,E1 -2976.499,E2 -2976.499} C_VEL
LIN {X 0,Y 558.95,Z 539.42,A -85,B 0,C 180,E1 -2977.95,E2 -2977.95} C_VEL
LIN {X 0,Y 559.005,Z 531.644,A -85,B 0,C 180,E1 -2979.407,E2 -2979.407} C_VEL
LIN {X 0,Y 559.218,Z 523.367,A -85,B 0,C 180,E1 -2980.683,E2 -2980.683} C_VEL
LIN {X 0,Y 559.362,Z 513.39,A -85,B 0,C 180,E1 -2981.965,E2 -2981.965} C_VEL
LIN {X 0,Y 559.596,Z 503.185,A -85,B 0,C 180,E1 -2983.065,E2 -2983.065} C_VEL
LIN {X 0,Y 559.862,Z 491.018,A -85,B 0,C 180,E1 -2984.169,E2 -2984.169} C_VEL
LIN {X 0,Y 560.125,Z 478.684,A -85,B 0,C 180,E1 -2985.1,E2 -2985.1} C_VEL
LIN {X 0,Y 560.391,Z 465.506,A -85,B 0,C 180,E1 -2985.923,E2 -2985.923} C_VEL
LIN {X 0,Y 560.674,Z 450.822,A -85,B 0,C 180,E1 -2986.663,E2 -2986.663} C_VEL
LIN {X 0,Y 560.934,Z 436.613,A -85,B 0,C 180,E1 -2987.218,E2 -2987.218} C_VEL
LIN {X 0,Y 561.129,Z 421.992,A -85,B 0,C 180,E1 -2987.642,E2 -2987.642} C_VEL
LIN {X 0,Y 561.248,Z 407.401,A -85,B 0,C 180,E1 -2987.926,E2 -2987.926} C_VEL
LIN {X 0,Y 561.754,Z 252.147,A -85,B 0,C 180,E1 -2989.97,E2 -2989.97} C_VEL
LIN {X 0,Y 560.466,Z 244.926,A -85,B 0,C 180,E1 -2990.133,E2 -2990.133} C_VEL
LIN {X 0,Y 560.841,Z 218.947,A -85,B 0,C 180,E1 -2992.859,E2 -2992.859} C_VEL
LIN {X 0,Y 561.406,Z 192.167,A -85,B 0,C 180,E1 -2995.752,E2 -2995.752} C_VEL
LIN {X 0,Y 559.542,Z 184.168,A -85,B 0,C 180,E1 -2996.726,E2 -2996.726} C_VEL
LIN {X 0,Y 559.157,Z 182.528,A -85,B 0,C 180,E1 -2996.979,E2 -2996.979} C_VEL
LIN {X 0,Y 559.117,Z 182.429,A -85,B 0,C 180,E1 -2999.852,E2 -2999.852} C_VEL
LIN {X 0,Y 559.149,Z 182.458,A -85,B 0,C 180,E1 -3002.716,E2 -3002.716} C_VEL
LIN {X 0,Y 559.125,Z 182.46,A -85,B 0,C 180,E1 -3005.324,E2 -3005.324} C_VEL
LIN {X 0,Y 559.128,Z 182.458,A -85,B 0,C 180,E1 -3008.018,E2 -3008.018} C_VEL
LIN {X 0,Y 559.153,Z 182.456,A -85,B 0,C 180,E1 -3010.812,E2 -3010.812} C_VEL
LIN {X 0,Y 559.135,Z 182.456,A -85,B 0,C 180,E1 -3013.734,E2 -3013.734} C_VEL
LIN {X 0,Y 559.142,Z 182.462,A -85,B 0,C 180,E1 -3016.804,E2 -3016.804} C_VEL
LIN {X 0,Y 559.153,Z 182.457,A -85,B 0,C 180,E1 -3019.187,E2 -3019.187} C_VEL
LIN {X 0,Y 559.129,Z 182.458,A -85,B 0,C 180,E1 -3021.982,E2 -3021.982} C_VEL
LIN {X 0,Y 559.131,Z 182.462,A -85,B 0,C 180,E1 -3024.787,E2 -3024.787} C_VEL
LIN {X 0,Y 559.153,Z 182.45,A -85,B 0,C 180,E1 -3027.364,E2 -3027.364} C_VEL
LIN {X 0,Y 559.142,Z 182.462,A -85,B 0,C 180,E1 -3030.143,E2 -3030.143} C_VEL
LIN {X 0,Y 559.168,Z 182.447,A -85,B 0,C 180,E1 -3033.172,E2 -3033.172} C_VEL
LIN {X 0,Y 559.153,Z 182.454,A -85,B 0,C 180,E1 -3035.495,E2 -3035.495} C_VEL
LIN {X 0,Y 559.167,Z 182.455,A -85,B 0,C 180,E1 -3038.624,E2 -3038.624} C_VEL
LIN {X 0,Y 559.161,Z 182.453,A -85,B 0,C 180,E1 -3040.926,E2 -3040.926} C_VEL
LIN {X 0,Y 559.16,Z 182.462,A -85,B 0,C 180,E1 -3043.948,E2 -3043.948} C_VEL
LIN {X 0,Y 559.17,Z 182.458,A -85,B 0,C 180,E1 -3046.184,E2 -3046.184} C_VEL
LIN {X 0,Y 559.19,Z 182.45,A -85,B 0,C 180,E1 -3049.134,E2 -3049.134} C_VEL
LIN {X 0,Y 559.201,Z 182.454,A -85,B 0,C 180,E1 -3052.054,E2 -3052.054} C_VEL
LIN {X 0,Y 559.249,Z 182.441,A -85,B 0,C 180,E1 -3054.953,E2 -3054.953} C_VEL
LIN {X 0,Y 559.247,Z 182.448,A -85,B 0,C 180,E1 -3057.84,E2 -3057.84} C_VEL
LIN {X 0,Y 559.269,Z 182.44,A -85,B 0,C 180,E1 -3060.72,E2 -3060.72} C_VEL
LIN {X 0,Y 559.237,Z 182.444,A -85,B 0,C 180,E1 -3062.882,E2 -3062.882} C_VEL
LIN {X 0,Y 559.225,Z 182.45,A -85,B 0,C 180,E1 -3065.77,E2 -3065.77} C_VEL
LIN {X 0,Y 559.189,Z 182.45,A -85,B 0,C 180,E1 -3068.675,E2 -3068.675} C_VEL
LIN {X 0,Y 559.203,Z 182.453,A -85,B 0,C 180,E1 -3071.601,E2 -3071.601} C_VEL
LIN {X 0,Y 559.197,Z 182.45,A -85,B 0,C 180,E1 -3074.596,E2 -3074.596} C_VEL
LIN {X 0,Y 559.157,Z 182.458,A -85,B 0,C 180,E1 -3077.557,E2 -3077.557} C_VEL
LIN {X 0,Y 559.17,Z 182.452,A -85,B 0,C 180,E1 -3079.838,E2 -3079.838} C_VEL
LIN {X 0,Y 559.139,Z 182.456,A -85,B 0,C 180,E1 -3082.153,E2 -3082.153} C_VEL
LIN {X 0,Y 559.174,Z 182.457,A -85,B 0,C 180,E1 -3085.298,E2 -3085.298} C_VEL
LIN {X 0,Y 559.155,Z 182.451,A -85,B 0,C 180,E1 -3087.714,E2 -3087.714} C_VEL
LIN {X 0,Y 559.138,Z 182.458,A -85,B 0,C 180,E1 -3090.62,E2 -3090.62} C_VEL
LIN {X 0,Y 558.477,Z 182.546,A -85,B 0,C 180,E1 -3091.221,E2 -3091.221} C_VEL
LIN {X 0,Y 555.613,Z 182.901,A -85,B 0,C 180,E1 -3092.197,E2 -3092.197} C_VEL
LIN {X 0,Y 553.202,Z 183.201,A -85,B 0,C 180,E1 -3092.983,E2 -3092.983} C_VEL
LIN {X 0,Y 552.185,Z 183.321,A -85,B 0,C 180,E1 -3093.59,E2 -3093.59} C_VEL
LIN {X 0,Y 552.112,Z 183.329,A -85,B 0,C 180,E1 -3093.795,E2 -3093.795} C_VEL
LIN {X 0,Y 552.112,Z 183.34,A -85,B 0,C 180,E1 -3096.747,E2 -3096.747} C_VEL
LIN {X 0,Y 552.129,Z 183.326,A -85,B 0,C 180,E1 -3099.527,E2 -3099.527} C_VEL
LIN {X 0,Y 552.129,Z 183.336,A -85,B 0,C 180,E1 -3102.426,E2 -3102.426} C_VEL
LIN {X 0,Y 552.096,Z 183.334,A -85,B 0,C 180,E1 -3105.563,E2 -3105.563} C_VEL
LIN {X 0,Y 552.133,Z 183.337,A -85,B 0,C 180,E1 -3108.556,E2 -3108.556} C_VEL
LIN {X 0,Y 552.116,Z 183.331,A -85,B 0,C 180,E1 -3111.411,E2 -3111.411} C_VEL
LIN {X 0,Y 552.1,Z 183.339,A -85,B 0,C 180,E1 -3114.158,E2 -3114.158} C_VEL
LIN {X 0,Y 552.117,Z 183.33,A -85,B 0,C 180,E1 -3116.814,E2 -3116.814} C_VEL
LIN {X 0,Y 552.103,Z 183.334,A -85,B 0,C 180,E1 -3119.391,E2 -3119.391} C_VEL
LIN {X 0,Y 552.08,Z 183.344,A -85,B 0,C 180,E1 -3121.9,E2 -3121.9} C_VEL
LIN {X 0,Y 552.173,Z 183.562,A -85,B 0,C 180,E1 -3124.282,E2 -3124.282} C_VEL
LIN {X 0,Y 553.857,Z 191.215,A -85,B 0,C 180,E1 -3125.445,E2 -3125.445} C_VEL
LIN {X 0,Y 553.614,Z 205.634,A -85,B 0,C 180,E1 -3127.417,E2 -3127.417} C_VEL
LIN {X 0,Y 553.176,Z 225.409,A -85,B 0,C 180,E1 -3130.078,E2 -3130.078} C_VEL
LIN {X 0,Y 552.886,Z 244.403,A -85,B 0,C 180,E1 -3132.576,E2 -3132.576} C_VEL
LIN {X 0,Y 554.273,Z 252.368,A -85,B 0,C 180,E1 -3132.759,E2 -3132.759} C_VEL
LIN {X 0,Y 553.785,Z 382.658,A -85,B 0,C 180,E1 -3134.496,E2 -3134.496} C_VEL
LIN {X 0,Y 553.615,Z 396.997,A -85,B 0,C 180,E1 -3134.84,E2 -3134.84} C_VEL
LIN {X 0,Y 553.368,Z 411.007,A -85,B 0,C 180,E1 -3135.332,E2 -3135.332} C_VEL
LIN {X 0,Y 553.168,Z 423.869,A -85,B 0,C 180,E1 -3135.937,E2 -3135.937} C_VEL
LIN {X 0,Y 552.913,Z 436.415,A -85,B 0,C 180,E1 -3136.68,E2 -3136.68} C_VEL
LIN {X 0,Y 552.641,Z 447.914,A -85,B 0,C 180,E1 -3137.514,E2 -3137.514} C_VEL
LIN {X 0,Y 552.45,Z 457.977,A -85,B 0,C 180,E1 -3138.395,E2 -3138.395} C_VEL
LIN {X 0,Y 552.286,Z 467.31,A -85,B 0,C 180,E1 -3139.367,E2 -3139.367} C_VEL
LIN {X 0,Y 552.075,Z 476.226,A -85,B 0,C 180,E1 -3140.474,E2 -3140.474} C_VEL
LIN {X 0,Y 551.928,Z 484.762,A -85,B 0,C 180,E1 -3141.764,E2 -3141.764} C_VEL
LIN {X 0,Y 551.824,Z 491.642,A -85,B 0,C 180,E1 -3143.051,E2 -3143.051} C_VEL
LIN {X 0,Y 551.792,Z 497.803,A -85,B 0,C 180,E1 -3144.518,E2 -3144.518} C_VEL
LIN {X 0,Y 551.76,Z 501.316,A -85,B 0,C 180,E1 -3145.617,E2 -3145.617} C_VEL
LIN {X 0,Y 551.72,Z 504.749,A -85,B 0,C 180,E1 -3147.079,E2 -3147.079} C_VEL
LIN {X 0,Y 551.643,Z 506.789,A -85,B 0,C 180,E1 -3148.54,E2 -3148.54} C_VEL
LIN {X 0,Y 551.64,Z 507.496,A -85,B 0,C 180,E1 -3150,E2 -3150} C_VEL
LIN {X 0,Y 551.641,Z 506.882,A -85,B 0,C 180,E1 -3151.46,E2 -3151.46} C_VEL
LIN {X 0,Y 551.719,Z 504.926,A -85,B 0,C 180,E1 -3152.92,E2 -3152.92} C_VEL
LIN {X 0,Y 551.761,Z 501.579,A -85,B 0,C 180,E1 -3154.383,E2 -3154.383} C_VEL
LIN {X 0,Y 551.819,Z 496.743,A -85,B 0,C 180,E1 -3155.848,E2 -3155.848} C_VEL
LIN {X 0,Y 551.833,Z 490.278,A -85,B 0,C 180,E1 -3157.317,E2 -3157.317} C_VEL
LIN {X 0,Y 551.959,Z 483.075,A -85,B 0,C 180,E1 -3158.604,E2 -3158.604} C_VEL
LIN {X 0,Y 552.067,Z 475.533,A -85,B 0,C 180,E1 -3159.71,E2 -3159.71} C_VEL
LIN {X 0,Y 552.282,Z 466.476,A -85,B 0,C 180,E1 -3160.818,E2 -3160.818} C_VEL
LIN {X 0,Y 552.468,Z 457.462,A -85,B 0,C 180,E1 -3161.743,E2 -3161.743} C_VEL
LIN {X 0,Y 552.658,Z 446.706,A -85,B 0,C 180,E1 -3162.671,E2 -3162.671} C_VEL
LIN {X 0,Y 552.919,Z 434.956,A -85,B 0,C 180,E1 -3163.506,E2 -3163.506} C_VEL
LIN {X 0,Y 553.233,Z 422.049,A -85,B 0,C 180,E1 -3164.248,E2 -3164.248} C_VEL
LIN {X 0,Y 553.495,Z 408.789,A -85,B 0,C 180,E1 -3164.847,E2 -3164.847} C_VEL
LIN {X 0,Y 553.676,Z 394.854,A -85,B 0,C 180,E1 -3165.312,E2 -3165.312} C_VEL
LIN {X 0,Y 553.784,Z 381.076,A -85,B 0,C 180,E1 -3165.621,E2 -3165.621} C_VEL
LIN {X 0,Y 554.285,Z 253.09,A -85,B 0,C 180,E1 -3167.321,E2 -3167.321} C_VEL
LIN {X 0,Y 552.887,Z 244.551,A -85,B 0,C 180,E1 -3167.505,E2 -3167.505} C_VEL
LIN {X 0,Y 553.18,Z 226.033,A -85,B 0,C 180,E1 -3169.923,E2 -3169.923} C_VEL
LIN {X 0,Y 553.708,Z 203.424,A -85,B 0,C 180,E1 -3172.972,E2 -3172.972} C_VEL
LIN {X 0,Y 553.92,Z 191.869,A -85,B 0,C 180,E1 -3174.551,E2 -3174.551} C_VEL
LIN {X 0,Y 552.148,Z 183.436,A -85,B 0,C 180,E1 -3175.845,E2 -3175.845} C_VEL
LIN {X 0,Y 552.094,Z 183.337,A -85,B 0,C 180,E1 -3178.928,E2 -3178.928} C_VEL
LIN {X 0,Y 552.11,Z 183.337,A -85,B 0,C 180,E1 -3181.475,E2 -3181.475} C_VEL
LIN {X 0,Y 552.133,Z 183.333,A -85,B 0,C 180,E1 -3184.17,E2 -3184.17} C_VEL
LIN {X 0,Y 552.109,Z 183.331,A -85,B 0,C 180,E1 -3186.746,E2 -3186.746} C_VEL
LIN {X 0,Y 552.127,Z 183.336,A -85,B 0,C 180,E1 -3189.526,E2 -3189.526} C_VEL
LIN {X 0,Y 552.128,Z 183.328,A -85,B 0,C 180,E1 -3192.425,E2 -3192.425} C_VEL
LIN {X 0,Y 552.094,Z 183.339,A -85,B 0,C 180,E1 -3195.562,E2 -3195.562} C_VEL
LIN {X 0,Y 552.136,Z 183.33,A -85,B 0,C 180,E1 -3198.675,E2 -3198.675} C_VEL
LIN {X 0,Y 552.113,Z 183.339,A -85,B 0,C 180,E1 -3201.41,E2 -3201.41} C_VEL
LIN {X 0,Y 552.109,Z 183.331,A -85,B 0,C 180,E1 -3204.158,E2 -3204.158} C_VEL
LIN {X 0,Y 552.118,Z 183.332,A -85,B 0,C 180,E1 -3206.814,E2 -3206.814} C_VEL
LIN {X 0,Y 552.137,Z 183.326,A -85,B 0,C 180,E1 -3209.944,E2 -3209.944} C_VEL
LIN {X 0,Y 552.134,Z 183.333,A -85,B 0,C 180,E1 -3212.999,E2 -3212.999} C_VEL
LIN {X 0,Y 552.107,Z 183.339,A -85,B 0,C 180,E1 -3215.161,E2 -3215.161} C_VEL
LIN {X 0,Y 552.089,Z 183.336,A -85,B 0,C 180,E1 -3217.549,E2 -3217.549} C_VEL
LIN {X 0,Y 552.142,Z 183.328,A -85,B 0,C 180,E1 -3220.373,E2 -3220.373} C_VEL
LIN {X 0,Y 552.151,Z 183.332,A -85,B 0,C 180,E1 -3222.977,E2 -3222.977} C_VEL
LIN {X 0,Y 552.131,Z 183.33,A -85,B 0,C 180,E1 -3226.004,E2 -3226.004} C_VEL
LIN {X 0,Y 552.155,Z 183.331,A -85,B 0,C 180,E1 -3228.993,E2 -3228.993} C_VEL
LIN {X 0,Y 552.154,Z 183.327,A -85,B 0,C 180,E1 -3231.951,E2 -3231.951} C_VEL
LIN {X 0,Y 552.224,Z 183.321,A -85,B 0,C 180,E1 -3234.889,E2 -3234.889} C_VEL
LIN {X 0,Y 552.217,Z 183.318,A -85,B 0,C 180,E1 -3237.812,E2 -3237.812} C_VEL
LIN {X 0,Y 552.238,Z 183.318,A -85,B 0,C 180,E1 -3240.729,E2 -3240.729} C_VEL
LIN {X 0,Y 552.2,Z 183.322,A -85,B 0,C 180,E1 -3242.918,E2 -3242.918} C_VEL
LIN {X 0,Y 552.195,Z 183.323,A -85,B 0,C 180,E1 -3245.844,E2 -3245.844} C_VEL
LIN {X 0,Y 552.156,Z 183.327,A -85,B 0,C 180,E1 -3248.786,E2 -3248.786} C_VEL
LIN {X 0,Y 552.155,Z 183.33,A -85,B 0,C 180,E1 -3251.751,E2 -3251.751} C_VEL
LIN {X 0,Y 552.129,Z 183.33,A -85,B 0,C 180,E1 -3254.748,E2 -3254.748} C_VEL
LIN {X 0,Y 552.107,Z 183.338,A -85,B 0,C 180,E1 -3257.788,E2 -3257.788} C_VEL
LIN {X 0,Y 552.123,Z 183.336,A -85,B 0,C 180,E1 -3260.101,E2 -3260.101} C_VEL
LIN {X 0,Y 552.088,Z 183.336,A -85,B 0,C 180,E1 -3262.451,E2 -3262.451} C_VEL
LIN {X 0,Y 552.15,Z 183.329,A -85,B 0,C 180,E1 -3265.351,E2 -3265.351} C_VEL
LIN {X 0,Y 552.114,Z 183.335,A -85,B 0,C 180,E1 -3268.098,E2 -3268.098} C_VEL
LIN {X 0,Y 552.096,Z 183.333,A -85,B 0,C 180,E1 -3270.61,E2 -3270.61} C_VEL
LIN {X 0,Y 552.116,Z 183.329,A -85,B 0,C 180,E1 -3273.186,E2 -3273.186} C_VEL
LIN {X 0,Y 552.096,Z 183.337,A -85,B 0,C 180,E1 -3275.843,E2 -3275.843} C_VEL
LIN {X 0,Y 552.119,Z 183.333,A -85,B 0,C 180,E1 -3279.062,E2 -3279.062} C_VEL
LIN {X 0,Y 552.114,Z 183.336,A -85,B 0,C 180,E1 -3281.446,E2 -3281.446} C_VEL
LIN {X 0,Y 552.082,Z 183.336,A -85,B 0,C 180,E1 -3284.532,E2 -3284.532} C_VEL
LIN {X 0,Y 552.124,Z 183.334,A -85,B 0,C 180,E1 -3287.585,E2 -3287.585} C_VEL
LIN {X 0,Y 552.124,Z 183.322,A -85,B 0,C 180,E1 -3290.473,E2 -3290.473} C_VEL
LIN {X 0,Y 552.102,Z 183.336,A -85,B 0,C 180,E1 -3293.318,E2 -3293.318} C_VEL
LIN {X 0,Y 552.097,Z 183.335,A -85,B 0,C 180,E1 -3295.938,E2 -3295.938} C_VEL
LIN {X 0,Y 552.116,Z 183.325,A -85,B 0,C 180,E1 -3298.541,E2 -3298.541} C_VEL
LIN {X 0,Y 552.099,Z 183.321,A -85,B 0,C 180,E1 -3301.443,E2 -3301.443} C_VEL
LIN {X 0,Y 552.151,Z 183.562,A -85,B 0,C 180,E1 -3302.817,E2 -3302.817} C_VEL
LIN {X 0,Y 554.626,Z 193.906,A -85,B 0,C 180,E1 -3304.116,E2 -3304.116} C_VEL
LIN {X 0,Y 553.981,Z 222.421,A -85,B 0,C 180,E1 -3307.237,E2 -3307.237} C_VEL
LIN {X 0,Y 553.547,Z 244.748,A -85,B 0,C 180,E1 -3309.615,E2 -3309.615} C_VEL
LIN {X 0,Y 554.527,Z 250.59,A -85,B 0,C 180,E1 -3309.761,E2 -3309.761} C_VEL
LIN {X 0,Y 555.106,Z 254.972,A -85,B 0,C 180,E1 -3309.841,E2 -3309.841} C_VEL
LIN {X 0,Y 554.467,Z 412.556,A -85,B 0,C 180,E1 -3311.938,E2 -3311.938} C_VEL
LIN {X 0,Y 554.254,Z 428.408,A -85,B 0,C 180,E1 -3312.307,E2 -3312.307} C_VEL
LIN {X 0,Y 554.025,Z 443.044,A -85,B 0,C 180,E1 -3312.799,E2 -3312.799} C_VEL
LIN {X 0,Y 553.749,Z 456.793,A -85,B 0,C 180,E1 -3313.408,E2 -3313.408} C_VEL
LIN {X 0,Y 553.433,Z 470.262,A -85,B 0,C 180,E1 -3314.156,E2 -3314.156} C_VEL
LIN {X 0,Y 553.076,Z 484.152,A -85,B 0,C 180,E1 -3315.103,E2 -3315.103} C_VEL
LIN {X 0,Y 552.76,Z 496.36,A -85,B 0,C 180,E1 -3316.115,E2 -3316.115} C_VEL
LIN {X 0,Y 552.481,Z 508.512,A -85,B 0,C 180,E1 -3317.325,E2 -3317.325} C_VEL
LIN {X 0,Y 552.215,Z 518.487,A -85,B 0,C 180,E1 -3318.514,E2 -3318.514} C_VEL
LIN {X 0,Y 552.124,Z 527.088,A -85,B 0,C 180,E1 -3319.735,E2 -3319.735} C_VEL
LIN {X 0,Y 551.92,Z 534.744,A -85,B 0,C 180,E1 -3321.026,E2 -3321.026} C_VEL
LIN {X 0,Y 551.837,Z 541.091,A -85,B 0,C 180,E1 -3322.316,E2 -3322.316} C_VEL
LIN {X 0,Y 551.769,Z 546.57,A -85,B 0,C 180,E1 -3323.681,E2 -3323.681} C_VEL
LIN {X 0,Y 551.713,Z 550.388,A -85,B 0,C 180,E1 -3324.885,E2 -3324.885} C_VEL
LIN {X 0,Y 551.73,Z 553.889,A -85,B 0,C 180,E1 -3326.349,E2 -3326.349} C_VEL
LIN {X 0,Y 551.655,Z 556.19,A -85,B 0,C 180,E1 -3327.81,E2 -3327.81} C_VEL
LIN {X 0,Y 551.639,Z 557.348,A -85,B 0,C 180,E1 -3329.27,E2 -3329.27} C_VEL
LIN {X 0,Y 551.639,Z 557.347,A -85,B 0,C 180,E1 -3330.73,E2 -3330.73} C_VEL
LIN {X 0,Y 551.655,Z 556.187,A -85,B 0,C 180,E1 -3332.191,E2 -3332.191} C_VEL
LIN {X 0,Y 551.73,Z 553.884,A -85,B 0,C 180,E1 -3333.652,E2 -3333.652} C_VEL
LIN {X 0,Y 551.713,Z 550.386,A -85,B 0,C 180,E1 -3335.116,E2 -3335.116} C_VEL
LIN {X 0,Y 551.82,Z 545.608,A -85,B 0,C 180,E1 -3336.582,E2 -3336.582} C_VEL
LIN {X 0,Y 551.876,Z 539.42,A -85,B 0,C 180,E1 -3338.053,E2 -3338.053} C_VEL
LIN {X 0,Y 551.95,Z 531.643,A -85,B 0,C 180,E1 -3339.528,E2 -3339.528} C_VEL
LIN {X 0,Y 552.184,Z 523.366,A -85,B 0,C 180,E1 -3340.821,E2 -3340.821} C_VEL
LIN {X 0,Y 552.352,Z 513.39,A -85,B 0,C 180,E1 -3342.119,E2 -3342.119} C_VEL
LIN {X 0,Y 552.609,Z 503.184,A -85,B 0,C 180,E1 -3343.234,E2 -3343.234} C_VEL
LIN {X 0,Y 552.907,Z 491.017,A -85,B 0,C 180,E1 -3344.351,E2 -3344.351} C_VEL
LIN {X 0,Y 553.254,Z 478.438,A -85,B 0,C 180,E1 -3345.31,E2 -3345.31} C_VEL
LIN {X 0,Y 553.546,Z 465.503,A -85,B 0,C 180,E1 -3346.125,E2 -3346.125} C_VEL
LIN {X 0,Y 553.852,Z 450.819,A -85,B 0,C 180,E1 -3346.874,E2 -3346.874} C_VEL
LIN {X 0,Y 554.15,Z 436.602,A -85,B 0,C 180,E1 -3347.435,E2 -3347.435} C_VEL
LIN {X 0,Y 554.35,Z 421.823,A -85,B 0,C 180,E1 -3347.864,E2 -3347.864} C_VEL
LIN {X 0,Y 554.497,Z 406.64,A -85,B 0,C 180,E1 -3348.156,E2 -3348.156} C_VEL
LIN {X 0,Y 555.038,Z 253.206,A -85,B 0,C 180,E1 -3350.185,E2 -3350.185} C_VEL
LIN {X 0,Y 553.553,Z 244.828,A -85,B 0,C 180,E1 -3350.38,E2 -3350.38} C_VEL
LIN {X 0,Y 554.027,Z 218.808,A -85,B 0,C 180,E1 -3353.156,E2 -3353.156} C_VEL
LIN {X 0,Y 554.634,Z 193.888,A -85,B 0,C 180,E1 -3355.885,E2 -3355.885} C_VEL
LIN {X 0,Y 552.143,Z 183.471,A -85,B 0,C 180,E1 -3357.206,E2 -3357.206} C_VEL
LIN {X 0,Y 552.093,Z 183.301,A -85,B 0,C 180,E1 -3360.046,E2 -3360.046} C_VEL
LIN {X 0,Y 552.107,Z 183.337,A -85,B 0,C 180,E1 -3362.845,E2 -3362.845} C_VEL
LIN {X 0,Y 552.074,Z 183.336,A -85,B 0,C 180,E1 -3365.439,E2 -3365.439} C_VEL
LIN {X 0,Y 552.092,Z 183.335,A -85,B 0,C 180,E1 -3367.885,E2 -3367.885} C_VEL
LIN {X 0,Y 552.106,Z 183.327,A -85,B 0,C 180,E1 -3370.481,E2 -3370.481} C_VEL
LIN {X 0,Y 552.105,Z 183.333,A -85,B 0,C 180,E1 -3373.424,E2 -3373.424} C_VEL
LIN {X 0,Y 552.104,Z 183.341,A -85,B 0,C 180,E1 -3376.576,E2 -3376.576} C_VEL
LIN {X 0,Y 552.107,Z 183.333,A -85,B 0,C 180,E1 -3379.519,E2 -3379.519} C_VEL
LIN {X 0,Y 552.089,Z 183.339,A -85,B 0,C 180,E1 -3382.336,E2 -3382.336} C_VEL
LIN {X 0,Y 552.083,Z 183.337,A -85,B 0,C 180,E1 -3385.051,E2 -3385.051} C_VEL
LIN {X 0,Y 552.113,Z 183.327,A -85,B 0,C 180,E1 -3387.681,E2 -3387.681} C_VEL
LIN {X 0,Y 552.105,Z 183.34,A -85,B 0,C 180,E1 -3390.235,E2 -3390.235} C_VEL
LIN {X 0,Y 552.136,Z 183.323,A -85,B 0,C 180,E1 -3393,E2 -3393} C_VEL
LIN {X 0,Y 552.11,Z 183.33,A -85,B 0,C 180,E1 -3395.161,E2 -3395.161} C_VEL
LIN {X 0,Y 552.122,Z 183.336,A -85,B 0,C 180,E1 -3398.337,E2 -3398.337} C_VEL
LIN {X 0,Y 552.149,Z 183.328,A -85,B 0,C 180,E1 -3400.674,E2 -3400.674} C_VEL
LIN {X 0,Y 552.11,Z 183.336,A -85,B 0,C 180,E1 -3403.737,E2 -3403.737} C_VEL
LIN {X 0,Y 552.133,Z 183.336,A -85,B 0,C 180,E1 -3406.005,E2 -3406.005} C_VEL
LIN {X 0,Y 552.158,Z 183.326,A -85,B 0,C 180,E1 -3408.993,E2 -3408.993} C_VEL
LIN {X 0,Y 552.155,Z 183.334,A -85,B 0,C 180,E1 -3411.952,E2 -3411.952} C_VEL
LIN {X 0,Y 552.224,Z 183.316,A -85,B 0,C 180,E1 -3414.889,E2 -3414.889} C_VEL
LIN {X 0,Y 552.219,Z 183.324,A -85,B 0,C 180,E1 -3417.812,E2 -3417.812} C_VEL
LIN {X 0,Y 552.24,Z 183.316,A -85,B 0,C 180,E1 -3420.729,E2 -3420.729} C_VEL
LIN {X 0,Y 552.204,Z 183.32,A -85,B 0,C 180,E1 -3422.918,E2 -3422.918} C_VEL
LIN {X 0,Y 552.196,Z 183.325,A -85,B 0,C 180,E1 -3425.844,E2 -3425.844} C_VEL
LIN {X 0,Y 552.159,Z 183.326,A -85,B 0,C 180,E1 -3428.786,E2 -3428.786} C_VEL
LIN {X 0,Y 552.16,Z 183.328,A -85,B 0,C 180,E1 -3431.751,E2 -3431.751} C_VEL
LIN {X 0,Y 552.134,Z 183.331,A -85,B 0,C 180,E1 -3434.749,E2 -3434.749} C_VEL
LIN {X 0,Y 552.107,Z 183.334,A -85,B 0,C 180,E1 -3437.789,E2 -3437.789} C_VEL
LIN {X 0,Y 552.129,Z 183.328,A -85,B 0,C 180,E1 -3440.101,E2 -3440.101} C_VEL
LIN {X 0,Y 552.091,Z 183.336,A -85,B 0,C 180,E1 -3442.451,E2 -3442.451} C_VEL
LIN {X 0,Y 552.154,Z 183.331,A -85,B 0,C 180,E1 -3445.351,E2 -3445.351} C_VEL
LIN {X 0,Y 552.108,Z 183.328,A -85,B 0,C 180,E1 -3448.099,E2 -3448.099} C_VEL
LIN {X 0,Y 552.101,Z 183.335,A -85,B 0,C 180,E1 -3450.616,E2 -3450.616} C_VEL
LIN {X 0,Y 552.114,Z 183.333,A -85,B 0,C 180,E1 -3453.186,E2 -3453.186} C_VEL
LIN {X 0,Y 552.112,Z 183.329,A -85,B 0,C 180,E1 -3453.795,E2 -3453.795} C_VEL
LIN {X 0,Y 551.481,Z 183.412,A -85,B 0,C 180,E1 -3454.404,E2 -3454.404} C_VEL
LIN {X 0,Y 548.661,Z 183.77,A -85,B 0,C 180,E1 -3455.392,E2 -3455.392} C_VEL
LIN {X 0,Y 546.239,Z 184.075,A -85,B 0,C 180,E1 -3456.187,E2 -3456.187} C_VEL
LIN {X 0,Y 545.167,Z 184.206,A -85,B 0,C 180,E1 -3456.801,E2 -3456.801} C_VEL
LIN {X 0,Y 545.065,Z 184.215,A -85,B 0,C 180,E1 -3457.009,E2 -3457.009} C_VEL
LIN {X 0,Y 545.065,Z 184.208,A -85,B 0,C 180,E1 -3460.143,E2 -3460.143} C_VEL
LIN {X 0,Y 545.078,Z 184.209,A -85,B 0,C 180,E1 -3463.107,E2 -3463.107} C_VEL
LIN {X 0,Y 545.057,Z 184.216,A -85,B 0,C 180,E1 -3466.226,E2 -3466.226} C_VEL
LIN {X 0,Y 545.088,Z 184.211,A -85,B 0,C 180,E1 -3468.886,E2 -3468.886} C_VEL
LIN {X 0,Y 545.051,Z 184.213,A -85,B 0,C 180,E1 -3471.763,E2 -3471.763} C_VEL
LIN {X 0,Y 545.052,Z 184.218,A -85,B 0,C 180,E1 -3474.533,E2 -3474.533} C_VEL
LIN {X 0,Y 545.07,Z 184.206,A -85,B 0,C 180,E1 -3477.212,E2 -3477.212} C_VEL
LIN {X 0,Y 545.064,Z 184.212,A -85,B 0,C 180,E1 -3479.811,E2 -3479.811} C_VEL
LIN {X 0,Y 545.053,Z 184.212,A -85,B 0,C 180,E1 -3482.342,E2 -3482.342} C_VEL
LIN {X 0,Y 545.131,Z 184.426,A -85,B 0,C 180,E1 -3484.034,E2 -3484.034} C_VEL
LIN {X 0,Y 547.146,Z 194.193,A -85,B 0,C 180,E1 -3485.528,E2 -3485.528} C_VEL
LIN {X 0,Y 546.585,Z 214.401,A -85,B 0,C 180,E1 -3488.305,E2 -3488.305} C_VEL
LIN {X 0,Y 546.12,Z 234.574,A -85,B 0,C 180,E1 -3491.038,E2 -3491.038} C_VEL
LIN {X 0,Y 545.985,Z 244.231,A -85,B 0,C 180,E1 -3492.314,E2 -3492.314} C_VEL
LIN {X 0,Y 546.5,Z 247.366,A -85,B 0,C 180,E1 -3492.414,E2 -3492.414} C_VEL
LIN {X 0,Y 547.594,Z 254.41,A -85,B 0,C 180,E1 -3492.548,E2 -3492.548} C_VEL
LIN {X 0,Y 547.038,Z 381.911,A -85,B 0,C 180,E1 -3494.252,E2 -3494.252} C_VEL
LIN {X 0,Y 546.856,Z 396.258,A -85,B 0,C 180,E1 -3494.586,E2 -3494.586} C_VEL
LIN {X 0,Y 546.682,Z 408.863,A -85,B 0,C 180,E1 -3495.017,E2 -3495.017} C_VEL
LIN {X 0,Y 546.441,Z 421.159,A -85,B 0,C 180,E1 -3495.57,E2 -3495.57} C_VEL
LIN {X 0,Y 546.076,Z 434.234,A -85,B 0,C 180,E1 -3496.321,E2 -3496.321} C_VEL
LIN {X 0,Y 545.813,Z 446.025,A -85,B 0,C 180,E1 -3497.167,E2 -3497.167} C_VEL
LIN {X 0,Y 545.514,Z 456.795,A -85,B 0,C 180,E1 -3498.104,E2 -3498.104} C_VEL
LIN {X 0,Y 545.285,Z 467.43,A -85,B 0,C 180,E1 -3499.229,E2 -3499.229} C_VEL
LIN {X 0,Y 545.031,Z 476.26,A -85,B 0,C 180,E1 -3500.35,E2 -3500.35} C_VEL
LIN {X 0,Y 544.874,Z 484.765,A -85,B 0,C 180,E1 -3501.656,E2 -3501.656} C_VEL
LIN {X 0,Y 544.737,Z 491.645,A -85,B 0,C 180,E1 -3502.96,E2 -3502.96} C_VEL
LIN {X 0,Y 544.724,Z 497.805,A -85,B 0,C 180,E1 -3504.447,E2 -3504.447} C_VEL
LIN {X 0,Y 544.655,Z 501.317,A -85,B 0,C 180,E1 -3505.559,E2 -3505.559} C_VEL
LIN {X 0,Y 544.647,Z 504.75,A -85,B 0,C 180,E1 -3507.041,E2 -3507.041} C_VEL
LIN {X 0,Y 544.544,Z 506.79,A -85,B 0,C 180,E1 -3508.521,E2 -3508.521} C_VEL
LIN {X 0,Y 544.54,Z 507.496,A -85,B 0,C 180,E1 -3510,E2 -3510} C_VEL
LIN {X 0,Y 544.542,Z 506.882,A -85,B 0,C 180,E1 -3511.479,E2 -3511.479} C_VEL
LIN {X 0,Y 544.646,Z 504.925,A -85,B 0,C 180,E1 -3512.958,E2 -3512.958} C_VEL
LIN {X 0,Y 544.655,Z 501.577,A -85,B 0,C 180,E1 -3514.44,E2 -3514.44} C_VEL
LIN {X 0,Y 544.73,Z 496.74,A -85,B 0,C 180,E1 -3515.924,E2 -3515.924} C_VEL
LIN {X 0,Y 544.783,Z 490.275,A -85,B 0,C 180,E1 -3517.412,E2 -3517.412} C_VEL
LIN {X 0,Y 544.905,Z 483.071,A -85,B 0,C 180,E1 -3518.716,E2 -3518.716} C_VEL
LIN {X 0,Y 545.079,Z 474.192,A -85,B 0,C 180,E1 -3520.024,E2 -3520.024} C_VEL
LIN {X 0,Y 545.345,Z 464.976,A -85,B 0,C 180,E1 -3521.145,E2 -3521.145} C_VEL
LIN {X 0,Y 545.576,Z 453.735,A -85,B 0,C 180,E1 -3522.271,E2 -3522.271} C_VEL
LIN {X 0,Y 545.878,Z 442.287,A -85,B 0,C 180,E1 -3523.21,E2 -3523.21} C_VEL
LIN {X 0,Y 546.224,Z 429.576,A -85,B 0,C 180,E1 -3524.055,E2 -3524.055} C_VEL
LIN {X 0,Y 546.5,Z 417.152,A -85,B 0,C 180,E1 -3524.713,E2 -3524.713} C_VEL
LIN {X 0,Y 546.766,Z 403.753,A -85,B 0,C 180,E1 -3525.261,E2 -3525.261} C_VEL
LIN {X 0,Y 546.981,Z 389.608,A -85,B 0,C 180,E1 -3525.677,E2 -3525.677} C_VEL
LIN {X 0,Y 547.08,Z 375.535,A -85,B 0,C 180,E1 -3525.937,E2 -3525.937} C_VEL
LIN {X 0,Y 547.564,Z 253.759,A -85,B 0,C 180,E1 -3527.552,E2 -3527.552} C_VEL
LIN {X 0,Y 545.963,Z 244.495,A -85,B 0,C 180,E1 -3527.757,E2 -3527.757} C_VEL
LIN {X 0,Y 546.39,Z 223.702,A -85,B 0,C 180,E1 -3530.518,E2 -3530.518} C_VEL
LIN {X 0,Y 546.956,Z 200.81,A -85,B 0,C 180,E1 -3533.647,E2 -3533.647} C_VEL
LIN {X 0,Y 547.07,Z 193.397,A -85,B 0,C 180,E1 -3534.677,E2 -3534.677} C_VEL
LIN {X 0,Y 545.105,Z 184.296,A -85,B 0,C 180,E1 -3536.101,E2 -3536.101} C_VEL
LIN {X 0,Y 545.057,Z 184.215,A -85,B 0,C 180,E1 -3539.338,E2 -3539.338} C_VEL
LIN {X 0,Y 545.054,Z 184.217,A -85,B 0,C 180,E1 -3541.914,E2 -3541.914} C_VEL
LIN {X 0,Y 545.075,Z 184.209,A -85,B 0,C 180,E1 -3544.563,E2 -3544.563} C_VEL
LIN {X 0,Y 545.037,Z 184.216,A -85,B 0,C 180,E1 -3547.303,E2 -3547.303} C_VEL
LIN {X 0,Y 545.063,Z 184.213,A -85,B 0,C 180,E1 -3550.142,E2 -3550.142} C_VEL
LIN {X 0,Y 545.076,Z 184.209,A -85,B 0,C 180,E1 -3553.106,E2 -3553.106} C_VEL
LIN {X 0,Y 545.046,Z 184.211,A -85,B 0,C 180,E1 -3556.225,E2 -3556.225} C_VEL
LIN {X 0,Y 545.093,Z 184.209,A -85,B 0,C 180,E1 -3558.886,E2 -3558.886} C_VEL
LIN {X 0,Y 545.048,Z 184.216,A -85,B 0,C 180,E1 -3561.762,E2 -3561.762} C_VEL
LIN {X 0,Y 545.06,Z 184.209,A -85,B 0,C 180,E1 -3564.533,E2 -3564.533} C_VEL
LIN {X 0,Y 545.076,Z 184.215,A -85,B 0,C 180,E1 -3567.212,E2 -3567.212} C_VEL
LIN {X 0,Y 545.097,Z 184.204,A -85,B 0,C 180,E1 -3569.812,E2 -3569.812} C_VEL
LIN {X 0,Y 545.09,Z 184.207,A -85,B 0,C 180,E1 -3572.825,E2 -3572.825} C_VEL
LIN {X 0,Y 545.046,Z 184.212,A -85,B 0,C 180,E1 -3575.63,E2 -3575.63} C_VEL
LIN {X 0,Y 545.06,Z 184.218,A -85,B 0,C 180,E1 -3578.836,E2 -3578.836} C_VEL
LIN {X 0,Y 545.077,Z 184.213,A -85,B 0,C 180,E1 -3581.195,E2 -3581.195} C_VEL
LIN {X 0,Y 545.07,Z 184.208,A -85,B 0,C 180,E1 -3583.521,E2 -3583.521} C_VEL
LIN {X 0,Y 545.089,Z 184.206,A -85,B 0,C 180,E1 -3585.82,E2 -3585.82} C_VEL
LIN {X 0,Y 545.111,Z 184.211,A -85,B 0,C 180,E1 -3588.849,E2 -3588.849} C_VEL
LIN {X 0,Y 545.124,Z 184.202,A -85,B 0,C 180,E1 -3591.847,E2 -3591.847} C_VEL
LIN {X 0,Y 545.199,Z 184.197,A -85,B 0,C 180,E1 -3594.823,E2 -3594.823} C_VEL
LIN {X 0,Y 545.189,Z 184.194,A -85,B 0,C 180,E1 -3597.784,E2 -3597.784} C_VEL
LIN {X 0,Y 545.208,Z 184.194,A -85,B 0,C 180,E1 -3600.738,E2 -3600.738} C_VEL
LIN {X 0,Y 545.167,Z 184.198,A -85,B 0,C 180,E1 -3602.956,E2 -3602.956} C_VEL
LIN {X 0,Y 545.166,Z 184.199,A -85,B 0,C 180,E1 -3605.919,E2 -3605.919} C_VEL
LIN {X 0,Y 545.114,Z 184.203,A -85,B 0,C 180,E1 -3608.9,E2 -3608.9} C_VEL
LIN {X 0,Y 545.127,Z 184.208,A -85,B 0,C 180,E1 -3611.904,E2 -3611.904} C_VEL
LIN {X 0,Y 545.078,Z 184.207,A -85,B 0,C 180,E1 -3614.944,E2 -3614.944} C_VEL
LIN {X 0,Y 545.074,Z 184.215,A -85,B 0,C 180,E1 -3618.026,E2 -3618.026} C_VEL
LIN {X 0,Y 545.087,Z 184.208,A -85,B 0,C 180,E1 -3620.372,E2 -3620.372} C_VEL
LIN {X 0,Y 545.084,Z 184.212,A -85,B 0,C 180,E1 -3623.559,E2 -3623.559} C_VEL
LIN {X 0,Y 545.082,Z 184.206,A -85,B 0,C 180,E1 -3626,E2 -3626} C_VEL
LIN {X 0,Y 545.081,Z 184.207,A -85,B 0,C 180,E1 -3628.748,E2 -3628.748} C_VEL
LIN {X 0,Y 545.052,Z 184.214,A -85,B 0,C 180,E1 -3631.679,E2 -3631.679} C_VEL
LIN {X 0,Y 545.073,Z 184.208,A -85,B 0,C 180,E1 -3634.564,E2 -3634.564} C_VEL
LIN {X 0,Y 545.031,Z 184.218,A -85,B 0,C 180,E1 -3637.304,E2 -3637.304} C_VEL
LIN {X 0,Y 545.062,Z 184.211,A -85,B 0,C 180,E1 -3640.143,E2 -3640.143} C_VEL
LIN {X 0,Y 545.072,Z 184.212,A -85,B 0,C 180,E1 -3643.107,E2 -3643.107} C_VEL
LIN {X 0,Y 545.043,Z 184.212,A -85,B 0,C 180,E1 -3646.227,E2 -3646.227} C_VEL
LIN {X 0,Y 545.076,Z 184.213,A -85,B 0,C 180,E1 -3648.886,E2 -3648.886} C_VEL
LIN {X 0,Y 545.043,Z 184.214,A -85,B 0,C 180,E1 -3651.865,E2 -3651.865} C_VEL
LIN {X 0,Y 545.031,Z 184.213,A -85,B 0,C 180,E1 -3654.532,E2 -3654.532} C_VEL
LIN {X 0,Y 545.059,Z 184.213,A -85,B 0,C 180,E1 -3657.212,E2 -3657.212} C_VEL
LIN {X 0,Y 545.058,Z 184.18,A -85,B 0,C 180,E1 -3659.811,E2 -3659.811} C_VEL
LIN {X 0,Y 545.1,Z 184.377,A -85,B 0,C 180,E1 -3662.533,E2 -3662.533} C_VEL
LIN {X 0,Y 547.863,Z 195.584,A -85,B 0,C 180,E1 -3663.977,E2 -3663.977} C_VEL
LIN {X 0,Y 547.145,Z 224.087,A -85,B 0,C 180,E1 -3667.136,E2 -3667.136} C_VEL
LIN {X 0,Y 546.657,Z 244.766,A -85,B 0,C 180,E1 -3669.369,E2 -3669.369} C_VEL
LIN {X 0,Y 547.767,Z 251.251,A -85,B 0,C 180,E1 -3669.531,E2 -3669.531} C_VEL
LIN {X 0,Y 548.371,Z 255.12,A -85,B 0,C 180,E1 -3669.606,E2 -3669.606} C_VEL
LIN {X 0,Y 547.64,Z 411.59,A -85,B 0,C 180,E1 -3671.721,E2 -3671.721} C_VEL
LIN {X 0,Y 547.459,Z 427.162,A -85,B 0,C 180,E1 -3672.08,E2 -3672.08} C_VEL
LIN {X 0,Y 547.198,Z 442.133,A -85,B 0,C 180,E1 -3672.578,E2 -3672.578} C_VEL
LIN {X 0,Y 546.851,Z 456.168,A -85,B 0,C 180,E1 -3673.193,E2 -3673.193} C_VEL
LIN {X 0,Y 546.545,Z 469.914,A -85,B 0,C 180,E1 -3673.951,E2 -3673.951} C_VEL
LIN {X 0,Y 546.136,Z 484.047,A -85,B 0,C 180,E1 -3674.91,E2 -3674.91} C_VEL
LIN {X 0,Y 545.817,Z 496.361,A -85,B 0,C 180,E1 -3675.935,E2 -3675.935} C_VEL
LIN {X 0,Y 545.511,Z 508.512,A -85,B 0,C 180,E1 -3677.16,E2 -3677.16} C_VEL
LIN {X 0,Y 545.174,Z 519.107,A -85,B 0,C 180,E1 -3678.446,E2 -3678.446} C_VEL
LIN {X 0,Y 545.05,Z 528.299,A -85,B 0,C 180,E1 -3679.788,E2 -3679.788} C_VEL
LIN {X 0,Y 544.845,Z 535.751,A -85,B 0,C 180,E1 -3681.096,E2 -3681.096} C_VEL
LIN {X 0,Y 544.744,Z 542.702,A -85,B 0,C 180,E1 -3682.588,E2 -3682.588} C_VEL
LIN {X 0,Y 544.709,Z 548.164,A -85,B 0,C 180,E1 -3684.076,E2 -3684.076} C_VEL
LIN {X 0,Y 544.605,Z 552.292,A -85,B 0,C 180,E1 -3685.56,E2 -3685.56} C_VEL
LIN {X 0,Y 544.644,Z 555.185,A -85,B 0,C 180,E1 -3687.042,E2 -3687.042} C_VEL
LIN {X 0,Y 544.544,Z 556.909,A -85,B 0,C 180,E1 -3688.521,E2 -3688.521} C_VEL
LIN {X 0,Y 544.538,Z 557.5,A -85,B 0,C 180,E1 -3690,E2 -3690} C_VEL
LIN {X 0,Y 544.544,Z 556.907,A -85,B 0,C 180,E1 -3691.479,E2 -3691.479} C_VEL
LIN {X 0,Y 544.644,Z 555.18,A -85,B 0,C 180,E1 -3692.959,E2 -3692.959} C_VEL
LIN {X 0,Y 544.605,Z 552.288,A -85,B 0,C 180,E1 -3694.441,E2 -3694.441} C_VEL
LIN {X 0,Y 544.709,Z 548.165,A -85,B 0,C 180,E1 -3695.925,E2 -3695.925} C_VEL
LIN {X 0,Y 544.745,Z 542.7,A -85,B 0,C 180,E1 -3697.413,E2 -3697.413} C_VEL
LIN {X 0,Y 544.845,Z 535.743,A -85,B 0,C 180,E1 -3698.905,E2 -3698.905} C_VEL
LIN {X 0,Y 545.074,Z 527.08,A -85,B 0,C 180,E1 -3700.4,E2 -3700.4} C_VEL
LIN {X 0,Y 545.237,Z 517.704,A -85,B 0,C 180,E1 -3701.735,E2 -3701.735} C_VEL
LIN {X 0,Y 545.511,Z 508.507,A -85,B 0,C 180,E1 -3702.841,E2 -3702.841} C_VEL
LIN {X 0,Y 545.828,Z 496.36,A -85,B 0,C 180,E1 -3704.066,E2 -3704.066} C_VEL
LIN {X 0,Y 546.137,Z 484.877,A -85,B 0,C 180,E1 -3705.027,E2 -3705.027} C_VEL
LIN {X 0,Y 546.476,Z 471.457,A -85,B 0,C 180,E1 -3705.956,E2 -3705.956} C_VEL
LIN {X 0,Y 546.82,Z 458.034,A -85,B 0,C 180,E1 -3706.713,E2 -3706.713} C_VEL
LIN {X 0,Y 547.133,Z 443.302,A -85,B 0,C 180,E1 -3707.377,E2 -3707.377} C_VEL
LIN {X 0,Y 547.428,Z 427.96,A -85,B 0,C 180,E1 -3707.898,E2 -3707.898} C_VEL
LIN {X 0,Y 547.61,Z 412.216,A -85,B 0,C 180,E1 -3708.268,E2 -3708.268} C_VEL
LIN {X 0,Y 548.327,Z 254.195,A -85,B 0,C 180,E1 -3710.408,E2 -3710.408} C_VEL
LIN {X 0,Y 546.739,Z 245.149,A -85,B 0,C 180,E1 -3710.606,E2 -3710.606} C_VEL
LIN {X 0,Y 546.916,Z 231.69,A -85,B 0,C 180,E1 -3712.034,E2 -3712.034} C_VEL
LIN {X 0,Y 547.573,Z 206.05,A -85,B 0,C 180,E1 -3714.856,E2 -3714.856} C_VEL
LIN {X 0,Y 547.799,Z 194.973,A -85,B 0,C 180,E1 -3716.095,E2 -3716.095} C_VEL
LIN {X 0,Y 545.102,Z 184.374,A -85,B 0,C 180,E1 -3717.467,E2 -3717.467} C_VEL
LIN {X 0,Y 545.041,Z 184.178,A -85,B 0,C 180,E1 -3720.24,E2 -3720.24} C_VEL
LIN {X 0,Y 545.071,Z 184.217,A -85,B 0,C 180,E1 -3723.061,E2 -3723.061} C_VEL
LIN {X 0,Y 545.031,Z 184.212,A -85,B 0,C 180,E1 -3725.673,E2 -3725.673} C_VEL
LIN {X 0,Y 545.048,Z 184.214,A -85,B 0,C 180,E1 -3728.237,E2 -3728.237} C_VEL
LIN {X 0,Y 545.079,Z 184.212,A -85,B 0,C 180,E1 -3731.115,E2 -3731.115} C_VEL
LIN {X 0,Y 545.046,Z 184.213,A -85,B 0,C 180,E1 -3734.13,E2 -3734.13} C_VEL
LIN {X 0,Y 545.06,Z 184.209,A -85,B 0,C 180,E1 -3737.303,E2 -3737.303} C_VEL
LIN {X 0,Y 545.065,Z 184.211,A -85,B 0,C 180,E1 -3739.857,E2 -3739.857} C_VEL
LIN {X 0,Y 545.067,Z 184.211,A -85,B 0,C 180,E1 -3743.074,E2 -3743.074} C_VEL
LIN {X 0,Y 545.063,Z 184.217,A -85,B 0,C 180,E1 -3746.328,E2 -3746.328} C_VEL
LIN {X 0,Y 545.063,Z 184.211,A -85,B 0,C 180,E1 -3748.952,E2 -3748.952} C_VEL
LIN {X 0,Y 545.081,Z 184.207,A -85,B 0,C 180,E1 -3751.507,E2 -3751.507} C_VEL
LIN {X 0,Y 545.093,Z 184.21,A -85,B 0,C 180,E1 -3754.491,E2 -3754.491} C_VEL
LIN {X 0,Y 545.034,Z 184.213,A -85,B 0,C 180,E1 -3757.242,E2 -3757.242} C_VEL
LIN {X 0,Y 545.114,Z 184.208,A -85,B 0,C 180,E1 -3760.415,E2 -3760.415} C_VEL
LIN {X 0,Y 545.061,Z 184.212,A -85,B 0,C 180,E1 -3763.521,E2 -3763.521} C_VEL
LIN {X 0,Y 545.092,Z 184.213,A -85,B 0,C 180,E1 -3765.82,E2 -3765.82} C_VEL
LIN {X 0,Y 545.114,Z 184.203,A -85,B 0,C 180,E1 -3768.849,E2 -3768.849} C_VEL
LIN {X 0,Y 545.125,Z 184.211,A -85,B 0,C 180,E1 -3771.847,E2 -3771.847} C_VEL
LIN {X 0,Y 545.2,Z 184.191,A -85,B 0,C 180,E1 -3774.823,E2 -3774.823} C_VEL
LIN {X 0,Y 545.191,Z 184.2,A -85,B 0,C 180,E1 -3777.784,E2 -3777.784} C_VEL
LIN {X 0,Y 545.21,Z 184.191,A -85,B 0,C 180,E1 -3780.739,E2 -3780.739} C_VEL
LIN {X 0,Y 545.17,Z 184.196,A -85,B 0,C 180,E1 -3782.956,E2 -3782.956} C_VEL
LIN {X 0,Y 545.167,Z 184.199,A -85,B 0,C 180,E1 -3785.92,E2 -3785.92} C_VEL
LIN {X 0,Y 545.118,Z 184.204,A -85,B 0,C 180,E1 -3788.9,E2 -3788.9} C_VEL
LIN {X 0,Y 545.133,Z 184.201,A -85,B 0,C 180,E1 -3791.904,E2 -3791.904} C_VEL
LIN {X 0,Y 545.083,Z 184.212,A -85,B 0,C 180,E1 -3794.944,E2 -3794.944} C_VEL
LIN {X 0,Y 545.075,Z 184.209,A -85,B 0,C 180,E1 -3798.026,E2 -3798.026} C_VEL
LIN {X 0,Y 545.093,Z 184.205,A -85,B 0,C 180,E1 -3800.372,E2 -3800.372} C_VEL
LIN {X 0,Y 545.079,Z 184.209,A -85,B 0,C 180,E1 -3803.56,E2 -3803.56} C_VEL
LIN {X 0,Y 545.078,Z 184.208,A -85,B 0,C 180,E1 -3806.001,E2 -3806.001} C_VEL
LIN {X 0,Y 545.088,Z 184.208,A -85,B 0,C 180,E1 -3808.748,E2 -3808.748} C_VEL
LIN {X 0,Y 545.056,Z 184.211,A -85,B 0,C 180,E1 -3811.679,E2 -3811.679} C_VEL
LIN {X 0,Y 545.081,Z 184.211,A -85,B 0,C 180,E1 -3814.563,E2 -3814.563} C_VEL
LIN {X 0,Y 545.065,Z 184.215,A -85,B 0,C 180,E1 -3817.009,E2 -3817.009} C_VEL
LIN {X 0,Y 544.355,Z 184.301,A -85,B 0,C 180,E1 -3817.626,E2 -3817.626} C_VEL
LIN {X 0,Y 541.488,Z 184.662,A -85,B 0,C 180,E1 -3818.626,E2 -3818.626} C_VEL
LIN {X 0,Y 539.1,Z 184.953,A -85,B 0,C 180,E1 -3819.432,E2 -3819.432} C_VEL
LIN {X 0,Y 538.091,Z 185.075,A -85,B 0,C 180,E1 -3820.054,E2 -3820.054} C_VEL
LIN {X 0,Y 538.016,Z 185.086,A -85,B 0,C 180,E1 -3820.265,E2 -3820.265} C_VEL
LIN {X 0,Y 538.025,Z 185.088,A -85,B 0,C 180,E1 -3822.988,E2 -3822.988} C_VEL
LIN {X 0,Y 538.024,Z 185.089,A -85,B 0,C 180,E1 -3825.926,E2 -3825.926} C_VEL
LIN {X 0,Y 538.05,Z 185.085,A -85,B 0,C 180,E1 -3829.225,E2 -3829.225} C_VEL
LIN {X 0,Y 537.992,Z 185.096,A -85,B 0,C 180,E1 -3832.122,E2 -3832.122} C_VEL
LIN {X 0,Y 538.012,Z 185.09,A -85,B 0,C 180,E1 -3834.917,E2 -3834.917} C_VEL
LIN {X 0,Y 538.02,Z 185.085,A -85,B 0,C 180,E1 -3837.618,E2 -3837.618} C_VEL
LIN {X 0,Y 538.015,Z 185.088,A -85,B 0,C 180,E1 -3840.239,E2 -3840.239} C_VEL
LIN {X 0,Y 538.033,Z 185.083,A -85,B 0,C 180,E1 -3842.795,E2 -3842.795} C_VEL
LIN {X 0,Y 538.08,Z 185.326,A -85,B 0,C 180,E1 -3843.784,E2 -3843.784} C_VEL
LIN {X 0,Y 540.33,Z 195.742,A -85,B 0,C 180,E1 -3845.404,E2 -3845.404} C_VEL
LIN {X 0,Y 539.697,Z 215.961,A -85,B 0,C 180,E1 -3848.215,E2 -3848.215} C_VEL
LIN {X 0,Y 539.196,Z 236.173,A -85,B 0,C 180,E1 -3850.983,E2 -3850.983} C_VEL
LIN {X 0,Y 539.077,Z 244.368,A -85,B 0,C 180,E1 -3852.072,E2 -3852.072} C_VEL
LIN {X 0,Y 540.8,Z 253.728,A -85,B 0,C 180,E1 -3852.29,E2 -3852.29} C_VEL
LIN {X 0,Y 540.324,Z 381.023,A -85,B 0,C 180,E1 -3854.003,E2 -3854.003} C_VEL
LIN {X 0,Y 540.152,Z 394.956,A -85,B 0,C 180,E1 -3854.316,E2 -3854.316} C_VEL
LIN {X 0,Y 539.913,Z 408.979,A -85,B 0,C 180,E1 -3854.788,E2 -3854.788} C_VEL
LIN {X 0,Y 539.622,Z 421.994,A -85,B 0,C 180,E1 -3855.384,E2 -3855.384} C_VEL
LIN {X 0,Y 539.221,Z 434.945,A -85,B 0,C 180,E1 -3856.143,E2 -3856.143} C_VEL
LIN {X 0,Y 538.923,Z 446.661,A -85,B 0,C 180,E1 -3857,E2 -3857} C_VEL
LIN {X 0,Y 538.604,Z 457.368,A -85,B 0,C 180,E1 -3857.949,E2 -3857.949} C_VEL
LIN {X 0,Y 538.329,Z 467.953,A -85,B 0,C 180,E1 -3859.088,E2 -3859.088} C_VEL
LIN {X 0,Y 538.039,Z 476.706,A -85,B 0,C 180,E1 -3860.223,E2 -3860.223} C_VEL
LIN {X 0,Y 537.841,Z 485.092,A -85,B 0,C 180,E1 -3861.546,E2 -3861.546} C_VEL
LIN {X 0,Y 537.692,Z 491.859,A -85,B 0,C 180,E1 -3862.867,E2 -3862.867} C_VEL
LIN {X 0,Y 537.655,Z 497.92,A -85,B 0,C 180,E1 -3864.374,E2 -3864.374} C_VEL
LIN {X 0,Y 537.553,Z 501.384,A -85,B 0,C 180,E1 -3865.501,E2 -3865.501} C_VEL
LIN {X 0,Y 537.547,Z 504.768,A -85,B 0,C 180,E1 -3867.002,E2 -3867.002} C_VEL
LIN {X 0,Y 537.45,Z 506.792,A -85,B 0,C 180,E1 -3868.501,E2 -3868.501} C_VEL
LIN {X 0,Y 537.441,Z 507.496,A -85,B 0,C 180,E1 -3870,E2 -3870} C_VEL
LIN {X 0,Y 537.448,Z 506.881,A -85,B 0,C 180,E1 -3871.498,E2 -3871.498} C_VEL
LIN {X 0,Y 537.546,Z 504.941,A -85,B 0,C 180,E1 -3872.997,E2 -3872.997} C_VEL
LIN {X 0,Y 537.552,Z 501.636,A -85,B 0,C 180,E1 -3874.499,E2 -3874.499} C_VEL
LIN {X 0,Y 537.643,Z 496.869,A -85,B 0,C 180,E1 -3876.002,E2 -3876.002} C_VEL
LIN {X 0,Y 537.727,Z 490.504,A -85,B 0,C 180,E1 -3877.51,E2 -3877.51} C_VEL
LIN {X 0,Y 537.867,Z 483.418,A -85,B 0,C 180,E1 -3878.831,E2 -3878.831} C_VEL
LIN {X 0,Y 538.091,Z 474.67,A -85,B 0,C 180,E1 -3880.155,E2 -3880.155} C_VEL
LIN {X 0,Y 538.391,Z 465.499,A -85,B 0,C 180,E1 -3881.291,E2 -3881.291} C_VEL
LIN {X 0,Y 538.619,Z 455.369,A -85,B 0,C 180,E1 -3882.337,E2 -3882.337} C_VEL
LIN {X 0,Y 538.977,Z 444.206,A -85,B 0,C 180,E1 -3883.286,E2 -3883.286} C_VEL
LIN {X 0,Y 539.33,Z 431.876,A -85,B 0,C 180,E1 -3884.142,E2 -3884.142} C_VEL
LIN {X 0,Y 539.669,Z 419.969,A -85,B 0,C 180,E1 -3884.807,E2 -3884.807} C_VEL
LIN {X 0,Y 539.974,Z 407.59,A -85,B 0,C 180,E1 -3885.352,E2 -3885.352} C_VEL
LIN {X 0,Y 540.186,Z 394.292,A -85,B 0,C 180,E1 -3885.79,E2 -3885.79} C_VEL
LIN {X 0,Y 540.301,Z 380.644,A -85,B 0,C 180,E1 -3886.094,E2 -3886.094} C_VEL
LIN {X 0,Y 540.874,Z 254.437,A -85,B 0,C 180,E1 -3887.788,E2 -3887.788} C_VEL
LIN {X 0,Y 539.065,Z 244.572,A -85,B 0,C 180,E1 -3888.006,E2 -3888.006} C_VEL
LIN {X 0,Y 539.374,Z 229.88,A -85,B 0,C 180,E1 -3889.965,E2 -3889.965} C_VEL
LIN {X 0,Y 540.027,Z 206.497,A -85,B 0,C 180,E1 -3893.183,E2 -3893.183} C_VEL
LIN {X 0,Y 540.224,Z 194.936,A -85,B 0,C 180,E1 -3894.806,E2 -3894.806} C_VEL
LIN {X 0,Y 538.051,Z 185.196,A -85,B 0,C 180,E1 -3896.343,E2 -3896.343} C_VEL
LIN {X 0,Y 538.029,Z 185.09,A -85,B 0,C 180,E1 -3898.933,E2 -3898.933} C_VEL
LIN {X 0,Y 538.009,Z 185.095,A -85,B 0,C 180,E1 -3901.886,E2 -3901.886} C_VEL
LIN {X 0,Y 538.025,Z 185.087,A -85,B 0,C 180,E1 -3904.619,E2 -3904.619} C_VEL
LIN {X 0,Y 538.005,Z 185.09,A -85,B 0,C 180,E1 -3907.17,E2 -3907.17} C_VEL
LIN {X 0,Y 538.021,Z 185.095,A -85,B 0,C 180,E1 -3909.796,E2 -3909.796} C_VEL
LIN {X 0,Y 538.016,Z 185.086,A -85,B 0,C 180,E1 -3912.785,E2 -3912.785} C_VEL
LIN {X 0,Y 538.017,Z 185.089,A -85,B 0,C 180,E1 -3915.926,E2 -3915.926} C_VEL
LIN {X 0,Y 538.048,Z 185.091,A -85,B 0,C 180,E1 -3919.224,E2 -3919.224} C_VEL
LIN {X 0,Y 537.988,Z 185.093,A -85,B 0,C 180,E1 -3922.122,E2 -3922.122} C_VEL
LIN {X 0,Y 538.015,Z 185.09,A -85,B 0,C 180,E1 -3924.917,E2 -3924.917} C_VEL
LIN {X 0,Y 538.021,Z 185.091,A -85,B 0,C 180,E1 -3927.617,E2 -3927.617} C_VEL
LIN {X 0,Y 538.038,Z 185.082,A -85,B 0,C 180,E1 -3930.24,E2 -3930.24} C_VEL
LIN {X 0,Y 538.06,Z 185.082,A -85,B 0,C 180,E1 -3932.796,E2 -3932.796} C_VEL
LIN {X 0,Y 538.043,Z 185.088,A -85,B 0,C 180,E1 -3935.292,E2 -3935.292} C_VEL
LIN {X 0,Y 538.009,Z 185.089,A -85,B 0,C 180,E1 -3938.041,E2 -3938.041} C_VEL
LIN {X 0,Y 538.034,Z 185.093,A -85,B 0,C 180,E1 -3940.94,E2 -3940.94} C_VEL
LIN {X 0,Y 538.021,Z 185.088,A -85,B 0,C 180,E1 -3943.299,E2 -3943.299} C_VEL
LIN {X 0,Y 538.058,Z 185.083,A -85,B 0,C 180,E1 -3945.63,E2 -3945.63} C_VEL
LIN {X 0,Y 538.07,Z 185.087,A -85,B 0,C 180,E1 -3948.701,E2 -3948.701} C_VEL
LIN {X 0,Y 538.081,Z 185.079,A -85,B 0,C 180,E1 -3951.739,E2 -3951.739} C_VEL
LIN {X 0,Y 538.157,Z 185.076,A -85,B 0,C 180,E1 -3954.755,E2 -3954.755} C_VEL
LIN {X 0,Y 538.161,Z 185.069,A -85,B 0,C 180,E1 -3957.755,E2 -3957.755} C_VEL
LIN {X 0,Y 538.177,Z 185.069,A -85,B 0,C 180,E1 -3960.748,E2 -3960.748} C_VEL
LIN {X 0,Y 538.133,Z 185.074,A -85,B 0,C 180,E1 -3962.994,E2 -3962.994} C_VEL
LIN {X 0,Y 538.119,Z 185.078,A -85,B 0,C 180,E1 -3965.997,E2 -3965.997} C_VEL
LIN {X 0,Y 538.065,Z 185.08,A -85,B 0,C 180,E1 -3969.018,E2 -3969.018} C_VEL
LIN {X 0,Y 538.076,Z 185.089,A -85,B 0,C 180,E1 -3972.063,E2 -3972.063} C_VEL
LIN {X 0,Y 538.038,Z 185.084,A -85,B 0,C 180,E1 -3975.144,E2 -3975.144} C_VEL
LIN {X 0,Y 538.026,Z 185.091,A -85,B 0,C 180,E1 -3978.27,E2 -3978.27} C_VEL
LIN {X 0,Y 538.031,Z 185.085,A -85,B 0,C 180,E1 -3980.652,E2 -3980.652} C_VEL
LIN {X 0,Y 538.017,Z 185.094,A -85,B 0,C 180,E1 -3983.888,E2 -3983.888} C_VEL
LIN {X 0,Y 538.043,Z 185.078,A -85,B 0,C 180,E1 -3986.366,E2 -3986.366} C_VEL
LIN {X 0,Y 538.022,Z 185.087,A -85,B 0,C 180,E1 -3988.934,E2 -3988.934} C_VEL
LIN {X 0,Y 538.007,Z 185.087,A -85,B 0,C 180,E1 -3991.888,E2 -3991.888} C_VEL
LIN {X 0,Y 538.023,Z 185.087,A -85,B 0,C 180,E1 -3994.621,E2 -3994.621} C_VEL
LIN {X 0,Y 538,Z 185.093,A -85,B 0,C 180,E1 -3997.171,E2 -3997.171} C_VEL
LIN {X 0,Y 538.019,Z 185.091,A -85,B 0,C 180,E1 -3999.797,E2 -3999.797} C_VEL
LIN {X 0,Y 538.012,Z 185.088,A -85,B 0,C 180,E1 -4002.787,E2 -4002.787} C_VEL
LIN {X 0,Y 538.012,Z 185.089,A -85,B 0,C 180,E1 -4005.927,E2 -4005.927} C_VEL
LIN {X 0,Y 538.025,Z 185.086,A -85,B 0,C 180,E1 -4008.227,E2 -4008.227} C_VEL
LIN {X 0,Y 538.006,Z 185.088,A -85,B 0,C 180,E1 -4011.17,E2 -4011.17} C_VEL
LIN {X 0,Y 537.99,Z 185.088,A -85,B 0,C 180,E1 -4014.089,E2 -4014.089} C_VEL
LIN {X 0,Y 538.027,Z 185.093,A -85,B 0,C 180,E1 -4016.728,E2 -4016.728} C_VEL
LIN {X 0,Y 538.002,Z 185.058,A -85,B 0,C 180,E1 -4019.561,E2 -4019.561} C_VEL
LIN {X 0,Y 538.059,Z 185.238,A -85,B 0,C 180,E1 -4022.255,E2 -4022.255} C_VEL
LIN {X 0,Y 541.084,Z 197.821,A -85,B 0,C 180,E1 -4023.9,E2 -4023.9} C_VEL
LIN {X 0,Y 540.307,Z 225.753,A -85,B 0,C 180,E1 -4027.032,E2 -4027.032} C_VEL
LIN {X 0,Y 539.823,Z 244.978,A -85,B 0,C 180,E1 -4029.133,E2 -4029.133} C_VEL
LIN {X 0,Y 541.676,Z 256.613,A -85,B 0,C 180,E1 -4029.385,E2 -4029.385} C_VEL
LIN {X 0,Y 540.813,Z 411.566,A -85,B 0,C 180,E1 -4031.516,E2 -4031.516} C_VEL
LIN {X 0,Y 540.607,Z 427.513,A -85,B 0,C 180,E1 -4031.894,E2 -4031.894} C_VEL
LIN {X 0,Y 540.309,Z 442.319,A -85,B 0,C 180,E1 -4032.397,E2 -4032.397} C_VEL
LIN {X 0,Y 539.961,Z 455.261,A -85,B 0,C 180,E1 -4032.972,E2 -4032.972} C_VEL
LIN {X 0,Y 539.636,Z 469.135,A -85,B 0,C 180,E1 -4033.74,E2 -4033.74} C_VEL
LIN {X 0,Y 539.279,Z 481.6,A -85,B 0,C 180,E1 -4034.583,E2 -4034.583} C_VEL
LIN {X 0,Y 538.904,Z 493.663,A -85,B 0,C 180,E1 -4035.558,E2 -4035.558} C_VEL
LIN {X 0,Y 538.585,Z 504.622,A -85,B 0,C 180,E1 -4036.608,E2 -4036.608} C_VEL
LIN {X 0,Y 538.305,Z 514.739,A -85,B 0,C 180,E1 -4037.752,E2 -4037.752} C_VEL
LIN {X 0,Y 538.111,Z 524.611,A -85,B 0,C 180,E1 -4039.084,E2 -4039.084} C_VEL
LIN {X 0,Y 537.824,Z 532.729,A -85,B 0,C 180,E1 -4040.41,E2 -4040.41} C_VEL
LIN {X 0,Y 537.734,Z 539.425,A -85,B 0,C 180,E1 -4041.735,E2 -4041.735} C_VEL
LIN {X 0,Y 537.618,Z 545.607,A -85,B 0,C 180,E1 -4043.244,E2 -4043.244} C_VEL
LIN {X 0,Y 537.574,Z 550.387,A -85,B 0,C 180,E1 -4044.75,E2 -4044.75} C_VEL
LIN {X 0,Y 537.561,Z 553.887,A -85,B 0,C 180,E1 -4046.252,E2 -4046.252} C_VEL
LIN {X 0,Y 537.488,Z 556.189,A -85,B 0,C 180,E1 -4047.752,E2 -4047.752} C_VEL
LIN {X 0,Y 537.44,Z 557.347,A -85,B 0,C 180,E1 -4049.251,E2 -4049.251} C_VEL
LIN {X 0,Y 537.44,Z 557.347,A -85,B 0,C 180,E1 -4050.75,E2 -4050.75} C_VEL
LIN {X 0,Y 537.488,Z 556.185,A -85,B 0,C 180,E1 -4052.248,E2 -4052.248} C_VEL
LIN {X 0,Y 537.561,Z 553.882,A -85,B 0,C 180,E1 -4053.748,E2 -4053.748} C_VEL
LIN {X 0,Y 537.574,Z 550.386,A -85,B 0,C 180,E1 -4055.251,E2 -4055.251} C_VEL
LIN {X 0,Y 537.664,Z 545.608,A -85,B 0,C 180,E1 -4056.756,E2 -4056.756} C_VEL
LIN {X 0,Y 537.734,Z 539.418,A -85,B 0,C 180,E1 -4058.266,E2 -4058.266} C_VEL
LIN {X 0,Y 537.859,Z 531.64,A -85,B 0,C 180,E1 -4059.78,E2 -4059.78} C_VEL
LIN {X 0,Y 538.102,Z 523.336,A -85,B 0,C 180,E1 -4061.107,E2 -4061.107} C_VEL
LIN {X 0,Y 538.335,Z 513.189,A -85,B 0,C 180,E1 -4062.44,E2 -4062.44} C_VEL
LIN {X 0,Y 538.653,Z 502.805,A -85,B 0,C 180,E1 -4063.583,E2 -4063.583} C_VEL
LIN {X 0,Y 538.992,Z 490.392,A -85,B 0,C 180,E1 -4064.73,E2 -4064.73} C_VEL
LIN {X 0,Y 539.387,Z 477.993,A -85,B 0,C 180,E1 -4065.681,E2 -4065.681} C_VEL
LIN {X 0,Y 539.734,Z 464.3,A -85,B 0,C 180,E1 -4066.549,E2 -4066.549} C_VEL
LIN {X 0,Y 540.138,Z 449.17,A -85,B 0,C 180,E1 -4067.316,E2 -4067.316} C_VEL
LIN {X 0,Y 540.478,Z 434.435,A -85,B 0,C 180,E1 -4067.891,E2 -4067.891} C_VEL
LIN {X 0,Y 540.718,Z 419.618,A -85,B 0,C 180,E1 -4068.314,E2 -4068.314} C_VEL
LIN {X 0,Y 540.878,Z 404.116,A -85,B 0,C 180,E1 -4068.603,E2 -4068.603} C_VEL
LIN {X 0,Y 541.682,Z 255.806,A -85,B 0,C 180,E1 -4070.626,E2 -4070.626} C_VEL
LIN {X 0,Y 539.835,Z 244.919,A -85,B 0,C 180,E1 -4070.872,E2 -4070.872} C_VEL
LIN {X 0,Y 540.39,Z 220.334,A -85,B 0,C 180,E1 -4073.573,E2 -4073.573} C_VEL
LIN {X 0,Y 541.108,Z 197.813,A -85,B 0,C 180,E1 -4076.1,E2 -4076.1} C_VEL
LIN {X 0,Y 538.061,Z 185.236,A -85,B 0,C 180,E1 -4077.746,E2 -4077.746} C_VEL
LIN {X 0,Y 538.005,Z 185.055,A -85,B 0,C 180,E1 -4080.628,E2 -4080.628} C_VEL
LIN {X 0,Y 538.018,Z 185.094,A -85,B 0,C 180,E1 -4083.278,E2 -4083.278} C_VEL
LIN {X 0,Y 537.992,Z 185.088,A -85,B 0,C 180,E1 -4086.004,E2 -4086.004} C_VEL
LIN {X 0,Y 538.009,Z 185.087,A -85,B 0,C 180,E1 -4088.831,E2 -4088.831} C_VEL
LIN {X 0,Y 538.028,Z 185.086,A -85,B 0,C 180,E1 -4091.773,E2 -4091.773} C_VEL
LIN {X 0,Y 538.002,Z 185.096,A -85,B 0,C 180,E1 -4094.862,E2 -4094.862} C_VEL
LIN {X 0,Y 538.016,Z 185.087,A -85,B 0,C 180,E1 -4097.214,E2 -4097.214} C_VEL
LIN {X 0,Y 538.022,Z 185.091,A -85,B 0,C 180,E1 -4100.203,E2 -4100.203} C_VEL
LIN {X 0,Y 538.021,Z 185.088,A -85,B 0,C 180,E1 -4103.067,E2 -4103.067} C_VEL
LIN {X 0,Y 538.016,Z 185.089,A -85,B 0,C 180,E1 -4105.827,E2 -4105.827} C_VEL
LIN {X 0,Y 538.006,Z 185.094,A -85,B 0,C 180,E1 -4108.499,E2 -4108.499} C_VEL
LIN {X 0,Y 538.016,Z 185.088,A -85,B 0,C 180,E1 -4111.097,E2 -4111.097} C_VEL
LIN {X 0,Y 538.039,Z 185.078,A -85,B 0,C 180,E1 -4113.633,E2 -4113.633} C_VEL
LIN {X 0,Y 538.004,Z 185.096,A -85,B 0,C 180,E1 -4116.122,E2 -4116.122} C_VEL
LIN {X 0,Y 538.035,Z 185.085,A -85,B 0,C 180,E1 -4119.349,E2 -4119.349} C_VEL
LIN {X 0,Y 538.051,Z 185.085,A -85,B 0,C 180,E1 -4122.517,E2 -4122.517} C_VEL
LIN {X 0,Y 538.061,Z 185.086,A -85,B 0,C 180,E1 -4125.631,E2 -4125.631} C_VEL
LIN {X 0,Y 538.073,Z 185.081,A -85,B 0,C 180,E1 -4128.702,E2 -4128.702} C_VEL
LIN {X 0,Y 538.082,Z 185.086,A -85,B 0,C 180,E1 -4131.74,E2 -4131.74} C_VEL
LIN {X 0,Y 538.157,Z 185.068,A -85,B 0,C 180,E1 -4134.755,E2 -4134.755} C_VEL
LIN {X 0,Y 538.163,Z 185.075,A -85,B 0,C 180,E1 -4137.755,E2 -4137.755} C_VEL
LIN {X 0,Y 538.18,Z 185.067,A -85,B 0,C 180,E1 -4140.748,E2 -4140.748} C_VEL
LIN {X 0,Y 538.137,Z 185.073,A -85,B 0,C 180,E1 -4142.995,E2 -4142.995} C_VEL
LIN {X 0,Y 538.121,Z 185.076,A -85,B 0,C 180,E1 -4145.997,E2 -4145.997} C_VEL
LIN {X 0,Y 538.068,Z 185.084,A -85,B 0,C 180,E1 -4149.018,E2 -4149.018} C_VEL
LIN {X 0,Y 538.081,Z 185.079,A -85,B 0,C 180,E1 -4152.063,E2 -4152.063} C_VEL
LIN {X 0,Y 538.043,Z 185.092,A -85,B 0,C 180,E1 -4155.144,E2 -4155.144} C_VEL
LIN {X 0,Y 538.028,Z 185.086,A -85,B 0,C 180,E1 -4158.27,E2 -4158.27} C_VEL
LIN {X 0,Y 538.038,Z 185.086,A -85,B 0,C 180,E1 -4160.652,E2 -4160.652} C_VEL
LIN {X 0,Y 538.002,Z 185.088,A -85,B 0,C 180,E1 -4163.889,E2 -4163.889} C_VEL
LIN {X 0,Y 538.04,Z 185.086,A -85,B 0,C 180,E1 -4166.367,E2 -4166.367} C_VEL
LIN {X 0,Y 538.029,Z 185.086,A -85,B 0,C 180,E1 -4168.934,E2 -4168.934} C_VEL
LIN {X 0,Y 538.008,Z 185.089,A -85,B 0,C 180,E1 -4171.887,E2 -4171.887} C_VEL
LIN {X 0,Y 538.031,Z 185.088,A -85,B 0,C 180,E1 -4174.621,E2 -4174.621} C_VEL
LIN {X 0,Y 538.007,Z 185.092,A -85,B 0,C 180,E1 -4177.171,E2 -4177.171} C_VEL
LIN {X 0,Y 538.016,Z 185.086,A -85,B 0,C 180,E1 -4180.265,E2 -4180.265} C_VEL
LIN {X 0,Y 537.366,Z 185.175,A -85,B 0,C 180,E1 -4180.89,E2 -4180.89} C_VEL
LIN {X 0,Y 534.512,Z 185.528,A -85,B 0,C 180,E1 -4181.905,E2 -4181.905} C_VEL
LIN {X 0,Y 532.086,Z 185.832,A -85,B 0,C 180,E1 -4182.722,E2 -4182.722} C_VEL
LIN {X 0,Y 531.038,Z 185.956,A -85,B 0,C 180,E1 -4183.353,E2 -4183.353} C_VEL
LIN {X 0,Y 530.951,Z 185.966,A -85,B 0,C 180,E1 -4183.567,E2 -4183.567} C_VEL
LIN {X 0,Y 530.96,Z 185.974,A -85,B 0,C 180,E1 -4186.505,E2 -4186.505} C_VEL
LIN {X 0,Y 530.987,Z 185.967,A -85,B 0,C 180,E1 -4188.976,E2 -4188.976} C_VEL
LIN {X 0,Y 530.956,Z 185.967,A -85,B 0,C 180,E1 -4191.529,E2 -4191.529} C_VEL
LIN {X 0,Y 530.963,Z 185.975,A -85,B 0,C 180,E1 -4194.381,E2 -4194.381} C_VEL
LIN {X 0,Y 530.968,Z 185.962,A -85,B 0,C 180,E1 -4197.134,E2 -4197.134} C_VEL
LIN {X 0,Y 530.97,Z 185.966,A -85,B 0,C 180,E1 -4199.803,E2 -4199.803} C_VEL
LIN {X 0,Y 530.975,Z 185.963,A -85,B 0,C 180,E1 -4202.476,E2 -4202.476} C_VEL
LIN {X 0,Y 531.027,Z 186.207,A -85,B 0,C 180,E1 -4203.523,E2 -4203.523} C_VEL
LIN {X 0,Y 533.494,Z 197.391,A -85,B 0,C 180,E1 -4205.288,E2 -4205.288} C_VEL
LIN {X 0,Y 532.817,Z 217.521,A -85,B 0,C 180,E1 -4208.122,E2 -4208.122} C_VEL
LIN {X 0,Y 532.28,Z 237.772,A -85,B 0,C 180,E1 -4210.926,E2 -4210.926} C_VEL
LIN {X 0,Y 532.186,Z 244.487,A -85,B 0,C 180,E1 -4211.819,E2 -4211.819} C_VEL
LIN {X 0,Y 534.18,Z 255.014,A -85,B 0,C 180,E1 -4212.059,E2 -4212.059} C_VEL
LIN {X 0,Y 533.59,Z 383.168,A -85,B 0,C 180,E1 -4213.796,E2 -4213.796} C_VEL
LIN {X 0,Y 533.358,Z 397.222,A -85,B 0,C 180,E1 -4214.137,E2 -4214.137} C_VEL
LIN {X 0,Y 533.108,Z 410.945,A -85,B 0,C 180,E1 -4214.629,E2 -4214.629} C_VEL
LIN {X 0,Y 532.823,Z 422.867,A -85,B 0,C 180,E1 -4215.193,E2 -4215.193} C_VEL
LIN {X 0,Y 532.374,Z 435.697,A -85,B 0,C 180,E1 -4215.961,E2 -4215.961} C_VEL
LIN {X 0,Y 532.051,Z 447.317,A -85,B 0,C 180,E1 -4216.829,E2 -4216.829} C_VEL
LIN {X 0,Y 531.688,Z 457.948,A -85,B 0,C 180,E1 -4217.79,E2 -4217.79} C_VEL
LIN {X 0,Y 531.366,Z 468.473,A -85,B 0,C 180,E1 -4218.943,E2 -4218.943} C_VEL
LIN {X 0,Y 531.046,Z 477.182,A -85,B 0,C 180,E1 -4220.093,E2 -4220.093} C_VEL
LIN {X 0,Y 530.821,Z 485.529,A -85,B 0,C 180,E1 -4221.434,E2 -4221.434} C_VEL
LIN {X 0,Y 530.641,Z 492.268,A -85,B 0,C 180,E1 -4222.772,E2 -4222.772} C_VEL
LIN {X 0,Y 530.585,Z 498.3,A -85,B 0,C 180,E1 -4224.298,E2 -4224.298} C_VEL
LIN {X 0,Y 530.48,Z 501.749,A -85,B 0,C 180,E1 -4225.441,E2 -4225.441} C_VEL
LIN {X 0,Y 530.482,Z 505.113,A -85,B 0,C 180,E1 -4226.962,E2 -4226.962} C_VEL
LIN {X 0,Y 530.36,Z 507.121,A -85,B 0,C 180,E1 -4228.481,E2 -4228.481} C_VEL
LIN {X 0,Y 530.349,Z 507.814,A -85,B 0,C 180,E1 -4230,E2 -4230} C_VEL
LIN {X 0,Y 530.358,Z 507.209,A -85,B 0,C 180,E1 -4231.518,E2 -4231.518} C_VEL
LIN {X 0,Y 530.481,Z 505.284,A -85,B 0,C 180,E1 -4233.037,E2 -4233.037} C_VEL
LIN {X 0,Y 530.48,Z 501.995,A -85,B 0,C 180,E1 -4234.559,E2 -4234.559} C_VEL
LIN {X 0,Y 530.588,Z 497.25,A -85,B 0,C 180,E1 -4236.082,E2 -4236.082} C_VEL
LIN {X 0,Y 530.688,Z 490.914,A -85,B 0,C 180,E1 -4237.61,E2 -4237.61} C_VEL
LIN {X 0,Y 530.846,Z 483.858,A -85,B 0,C 180,E1 -4238.949,E2 -4238.949} C_VEL
LIN {X 0,Y 531.12,Z 475.144,A -85,B 0,C 180,E1 -4240.29,E2 -4240.29} C_VEL
LIN {X 0,Y 531.447,Z 466.021,A -85,B 0,C 180,E1 -4241.441,E2 -4241.441} C_VEL
LIN {X 0,Y 531.755,Z 454.912,A -85,B 0,C 180,E1 -4242.595,E2 -4242.595} C_VEL
LIN {X 0,Y 532.136,Z 443.613,A -85,B 0,C 180,E1 -4243.557,E2 -4243.557} C_VEL
LIN {X 0,Y 532.552,Z 431.099,A -85,B 0,C 180,E1 -4244.423,E2 -4244.423} C_VEL
LIN {X 0,Y 532.916,Z 418.929,A -85,B 0,C 180,E1 -4245.097,E2 -4245.097} C_VEL
LIN {X 0,Y 533.231,Z 406.103,A -85,B 0,C 180,E1 -4245.651,E2 -4245.651} C_VEL
LIN {X 0,Y 533.471,Z 392.393,A -85,B 0,C 180,E1 -4246.085,E2 -4246.085} C_VEL
LIN {X 0,Y 533.627,Z 378.263,A -85,B 0,C 180,E1 -4246.375,E2 -4246.375} C_VEL
LIN {X 0,Y 534.175,Z 255.466,A -85,B 0,C 180,E1 -4248.026,E2 -4248.026} C_VEL
LIN {X 0,Y 532.185,Z 244.536,A -85,B 0,C 180,E1 -4248.269,E2 -4248.269} C_VEL
LIN {X 0,Y 532.694,Z 223.993,A -85,B 0,C 180,E1 -4251.07,E2 -4251.07} C_VEL
LIN {X 0,Y 533.376,Z 200.933,A -85,B 0,C 180,E1 -4254.299,E2 -4254.299} C_VEL
LIN {X 0,Y 533.354,Z 196.489,A -85,B 0,C 180,E1 -4254.939,E2 -4254.939} C_VEL
LIN {X 0,Y 530.988,Z 186.064,A -85,B 0,C 180,E1 -4256.613,E2 -4256.613} C_VEL
LIN {X 0,Y 530.979,Z 185.966,A -85,B 0,C 180,E1 -4259.322,E2 -4259.322} C_VEL
LIN {X 0,Y 530.964,Z 185.969,A -85,B 0,C 180,E1 -4262.1,E2 -4262.1} C_VEL
LIN {X 0,Y 530.982,Z 185.965,A -85,B 0,C 180,E1 -4264.853,E2 -4264.853} C_VEL
LIN {X 0,Y 530.964,Z 185.971,A -85,B 0,C 180,E1 -4267.507,E2 -4267.507} C_VEL
LIN {X 0,Y 530.979,Z 185.966,A -85,B 0,C 180,E1 -4270.432,E2 -4270.432} C_VEL
LIN {X 0,Y 530.961,Z 185.969,A -85,B 0,C 180,E1 -4273.281,E2 -4273.281} C_VEL
LIN {X 0,Y 530.98,Z 185.968,A -85,B 0,C 180,E1 -4275.621,E2 -4275.621} C_VEL
LIN {X 0,Y 530.996,Z 185.963,A -85,B 0,C 180,E1 -4278.564,E2 -4278.564} C_VEL
LIN {X 0,Y 530.953,Z 185.975,A -85,B 0,C 180,E1 -4281.529,E2 -4281.529} C_VEL
LIN {X 0,Y 530.977,Z 185.963,A -85,B 0,C 180,E1 -4284.382,E2 -4284.382} C_VEL
LIN {X 0,Y 530.965,Z 185.971,A -85,B 0,C 180,E1 -4287.133,E2 -4287.133} C_VEL
LIN {X 0,Y 530.981,Z 185.962,A -85,B 0,C 180,E1 -4289.804,E2 -4289.804} C_VEL
LIN {X 0,Y 531.01,Z 185.956,A -85,B 0,C 180,E1 -4292.466,E2 -4292.466} C_VEL
LIN {X 0,Y 531,Z 185.97,A -85,B 0,C 180,E1 -4294.942,E2 -4294.942} C_VEL
LIN {X 0,Y 530.965,Z 185.967,A -85,B 0,C 180,E1 -4298.246,E2 -4298.246} C_VEL
LIN {X 0,Y 530.991,Z 185.967,A -85,B 0,C 180,E1 -4300.677,E2 -4300.677} C_VEL
LIN {X 0,Y 530.986,Z 185.967,A -85,B 0,C 180,E1 -4303.071,E2 -4303.071} C_VEL
LIN {X 0,Y 531.012,Z 185.961,A -85,B 0,C 180,E1 -4305.436,E2 -4305.436} C_VEL
LIN {X 0,Y 531.029,Z 185.963,A -85,B 0,C 180,E1 -4308.549,E2 -4308.549} C_VEL
LIN {X 0,Y 531.05,Z 185.954,A -85,B 0,C 180,E1 -4311.629,E2 -4311.629} C_VEL
LIN {X 0,Y 531.116,Z 185.954,A -85,B 0,C 180,E1 -4314.685,E2 -4314.685} C_VEL
LIN {X 0,Y 531.133,Z 185.944,A -85,B 0,C 180,E1 -4317.725,E2 -4317.725} C_VEL
LIN {X 0,Y 531.147,Z 185.944,A -85,B 0,C 180,E1 -4320.758,E2 -4320.758} C_VEL
LIN {X 0,Y 531.1,Z 185.95,A -85,B 0,C 180,E1 -4323.034,E2 -4323.034} C_VEL
LIN {X 0,Y 531.078,Z 185.956,A -85,B 0,C 180,E1 -4326.077,E2 -4326.077} C_VEL
LIN {X 0,Y 531.025,Z 185.957,A -85,B 0,C 180,E1 -4329.138,E2 -4329.138} C_VEL
LIN {X 0,Y 531.033,Z 185.964,A -85,B 0,C 180,E1 -4332.225,E2 -4332.225} C_VEL
LIN {X 0,Y 530.988,Z 185.964,A -85,B 0,C 180,E1 -4335.35,E2 -4335.35} C_VEL
LIN {X 0,Y 530.985,Z 185.965,A -85,B 0,C 180,E1 -4338.521,E2 -4338.521} C_VEL
LIN {X 0,Y 530.992,Z 185.961,A -85,B 0,C 180,E1 -4340.938,E2 -4340.938} C_VEL
LIN {X 0,Y 530.973,Z 185.966,A -85,B 0,C 180,E1 -4344.225,E2 -4344.225} C_VEL
LIN {X 0,Y 531.004,Z 185.953,A -85,B 0,C 180,E1 -4346.744,E2 -4346.744} C_VEL
LIN {X 0,Y 530.973,Z 185.968,A -85,B 0,C 180,E1 -4349.323,E2 -4349.323} C_VEL
LIN {X 0,Y 530.963,Z 185.962,A -85,B 0,C 180,E1 -4352.102,E2 -4352.102} C_VEL
LIN {X 0,Y 530.979,Z 185.965,A -85,B 0,C 180,E1 -4354.854,E2 -4354.854} C_VEL
LIN {X 0,Y 530.96,Z 185.969,A -85,B 0,C 180,E1 -4357.508,E2 -4357.508} C_VEL
LIN {X 0,Y 530.975,Z 185.965,A -85,B 0,C 180,E1 -4360.433,E2 -4360.433} C_VEL
LIN {X 0,Y 530.955,Z 185.974,A -85,B 0,C 180,E1 -4363.282,E2 -4363.282} C_VEL
LIN {X 0,Y 530.97,Z 185.969,A -85,B 0,C 180,E1 -4365.623,E2 -4365.623} C_VEL
LIN {X 0,Y 530.988,Z 185.964,A -85,B 0,C 180,E1 -4368.565,E2 -4368.565} C_VEL
LIN {X 0,Y 530.951,Z 185.973,A -85,B 0,C 180,E1 -4371.53,E2 -4371.53} C_VEL
LIN {X 0,Y 530.949,Z 185.966,A -85,B 0,C 180,E1 -4374.38,E2 -4374.38} C_VEL
LIN {X 0,Y 530.962,Z 185.97,A -85,B 0,C 180,E1 -4377.134,E2 -4377.134} C_VEL
LIN {X 0,Y 530.949,Z 185.93,A -85,B 0,C 180,E1 -4379.803,E2 -4379.803} C_VEL
LIN {X 0,Y 531.004,Z 186.123,A -85,B 0,C 180,E1 -4381.976,E2 -4381.976} C_VEL
LIN {X 0,Y 534.278,Z 199.123,A -85,B 0,C 180,E1 -4383.71,E2 -4383.71} C_VEL
LIN {X 0,Y 533.55,Z 223.811,A -85,B 0,C 180,E1 -4386.519,E2 -4386.519} C_VEL
LIN {X 0,Y 532.991,Z 244.809,A -85,B 0,C 180,E1 -4388.864,E2 -4388.864} C_VEL
LIN {X 0,Y 534.564,Z 254.427,A -85,B 0,C 180,E1 -4389.091,E2 -4389.091} C_VEL
LIN {X 0,Y 534.97,Z 258.518,A -85,B 0,C 180,E1 -4389.164,E2 -4389.164} C_VEL
LIN {X 0,Y 533.994,Z 411.38,A -85,B 0,C 180,E1 -4391.303,E2 -4391.303} C_VEL
LIN {X 0,Y 533.751,Z 427.055,A -85,B 0,C 180,E1 -4391.678,E2 -4391.678} C_VEL
LIN {X 0,Y 533.424,Z 442.479,A -85,B 0,C 180,E1 -4392.212,E2 -4392.212} C_VEL
LIN {X 0,Y 533.049,Z 456.358,A -85,B 0,C 180,E1 -4392.843,E2 -4392.843} C_VEL
LIN {X 0,Y 532.687,Z 469.959,A -85,B 0,C 180,E1 -4393.62,E2 -4393.62} C_VEL
LIN {X 0,Y 532.251,Z 483.398,A -85,B 0,C 180,E1 -4394.56,E2 -4394.56} C_VEL
LIN {X 0,Y 531.806,Z 496.29,A -85,B 0,C 180,E1 -4395.654,E2 -4395.654} C_VEL
LIN {X 0,Y 531.476,Z 507.681,A -85,B 0,C 180,E1 -4396.815,E2 -4396.815} C_VEL
LIN {X 0,Y 531.119,Z 518.693,A -85,B 0,C 180,E1 -4398.161,E2 -4398.161} C_VEL
LIN {X 0,Y 530.946,Z 527.894,A -85,B 0,C 180,E1 -4399.514,E2 -4399.514} C_VEL
LIN {X 0,Y 530.738,Z 535.483,A -85,B 0,C 180,E1 -4400.857,E2 -4400.857} C_VEL
LIN {X 0,Y 530.6,Z 542.559,A -85,B 0,C 180,E1 -4402.389,E2 -4402.389} C_VEL
LIN {X 0,Y 530.528,Z 548.113,A -85,B 0,C 180,E1 -4403.917,E2 -4403.917} C_VEL
LIN {X 0,Y 530.412,Z 552.288,A -85,B 0,C 180,E1 -4405.44,E2 -4405.44} C_VEL
LIN {X 0,Y 530.449,Z 555.183,A -85,B 0,C 180,E1 -4406.962,E2 -4406.962} C_VEL
LIN {X 0,Y 530.359,Z 556.909,A -85,B 0,C 180,E1 -4408.482,E2 -4408.482} C_VEL
LIN {X 0,Y 530.34,Z 557.5,A -85,B 0,C 180,E1 -4410,E2 -4410} C_VEL
LIN {X 0,Y 530.359,Z 556.906,A -85,B 0,C 180,E1 -4411.519,E2 -4411.519} C_VEL
LIN {X 0,Y 530.449,Z 555.177,A -85,B 0,C 180,E1 -4413.038,E2 -4413.038} C_VEL
LIN {X 0,Y 530.412,Z 552.284,A -85,B 0,C 180,E1 -4414.56,E2 -4414.56} C_VEL
LIN {X 0,Y 530.533,Z 548.115,A -85,B 0,C 180,E1 -4416.084,E2 -4416.084} C_VEL
LIN {X 0,Y 530.601,Z 542.557,A -85,B 0,C 180,E1 -4417.612,E2 -4417.612} C_VEL
LIN {X 0,Y 530.739,Z 535.474,A -85,B 0,C 180,E1 -4419.143,E2 -4419.143} C_VEL
LIN {X 0,Y 530.96,Z 526.646,A -85,B 0,C 180,E1 -4420.679,E2 -4420.679} C_VEL
LIN {X 0,Y 531.19,Z 517.063,A -85,B 0,C 180,E1 -4422.051,E2 -4422.051} C_VEL
LIN {X 0,Y 531.477,Z 507.675,A -85,B 0,C 180,E1 -4423.186,E2 -4423.186} C_VEL
LIN {X 0,Y 531.815,Z 496.29,A -85,B 0,C 180,E1 -4424.346,E2 -4424.346} C_VEL
LIN {X 0,Y 532.206,Z 483.65,A -85,B 0,C 180,E1 -4425.422,E2 -4425.422} C_VEL
LIN {X 0,Y 532.636,Z 469.942,A -85,B 0,C 180,E1 -4426.382,E2 -4426.382} C_VEL
LIN {X 0,Y 533.054,Z 456.34,A -85,B 0,C 180,E1 -4427.158,E2 -4427.158} C_VEL
LIN {X 0,Y 533.458,Z 441.264,A -85,B 0,C 180,E1 -4427.837,E2 -4427.837} C_VEL
LIN {X 0,Y 533.778,Z 426.203,A -85,B 0,C 180,E1 -4428.346,E2 -4428.346} C_VEL
LIN {X 0,Y 534.03,Z 410.38,A -85,B 0,C 180,E1 -4428.713,E2 -4428.713} C_VEL
LIN {X 0,Y 534.982,Z 256.78,A -85,B 0,C 180,E1 -4430.861,E2 -4430.861} C_VEL
LIN {X 0,Y 533.01,Z 245,A -85,B 0,C 180,E1 -4431.124,E2 -4431.124} C_VEL
LIN {X 0,Y 533.581,Z 222,A -85,B 0,C 180,E1 -4433.686,E2 -4433.686} C_VEL
LIN {X 0,Y 534.328,Z 199.117,A -85,B 0,C 180,E1 -4436.288,E2 -4436.288} C_VEL
LIN {X 0,Y 531.004,Z 186.121,A -85,B 0,C 180,E1 -4438.024,E2 -4438.024} C_VEL
LIN {X 0,Y 530.959,Z 185.93,A -85,B 0,C 180,E1 -4440.642,E2 -4440.642} C_VEL
LIN {X 0,Y 530.961,Z 185.97,A -85,B 0,C 180,E1 -4443.5,E2 -4443.5} C_VEL
LIN {X 0,Y 530.953,Z 185.968,A -85,B 0,C 180,E1 -4446.558,E2 -4446.558} C_VEL
LIN {X 0,Y 530.969,Z 185.954,A -85,B 0,C 180,E1 -4449.445,E2 -4449.445} C_VEL
LIN {X 0,Y 530.976,Z 185.969,A -85,B 0,C 180,E1 -4452.457,E2 -4452.457} C_VEL
LIN {X 0,Y 530.973,Z 185.966,A -85,B 0,C 180,E1 -4455.622,E2 -4455.622} C_VEL
LIN {X 0,Y 530.991,Z 185.966,A -85,B 0,C 180,E1 -4458.564,E2 -4458.564} C_VEL
LIN {X 0,Y 530.954,Z 185.966,A -85,B 0,C 180,E1 -4461.529,E2 -4461.529} C_VEL
LIN {X 0,Y 530.952,Z 185.974,A -85,B 0,C 180,E1 -4464.38,E2 -4464.38} C_VEL
LIN {X 0,Y 530.964,Z 185.96,A -85,B 0,C 180,E1 -4467.133,E2 -4467.133} C_VEL
LIN {X 0,Y 530.965,Z 185.967,A -85,B 0,C 180,E1 -4469.803,E2 -4469.803} C_VEL
LIN {X 0,Y 531.011,Z 185.959,A -85,B 0,C 180,E1 -4472.467,E2 -4472.467} C_VEL
LIN {X 0,Y 530.992,Z 185.962,A -85,B 0,C 180,E1 -4474.942,E2 -4474.942} C_VEL
LIN {X 0,Y 530.968,Z 185.971,A -85,B 0,C 180,E1 -4478.247,E2 -4478.247} C_VEL
LIN {X 0,Y 530.991,Z 185.964,A -85,B 0,C 180,E1 -4480.677,E2 -4480.677} C_VEL
LIN {X 0,Y 530.978,Z 185.964,A -85,B 0,C 180,E1 -4483.071,E2 -4483.071} C_VEL
LIN {X 0,Y 531.016,Z 185.961,A -85,B 0,C 180,E1 -4485.436,E2 -4485.436} C_VEL
LIN {X 0,Y 531.033,Z 185.959,A -85,B 0,C 180,E1 -4488.55,E2 -4488.55} C_VEL
LIN {X 0,Y 531.052,Z 185.96,A -85,B 0,C 180,E1 -4491.63,E2 -4491.63} C_VEL
LIN {X 0,Y 531.117,Z 185.945,A -85,B 0,C 180,E1 -4494.685,E2 -4494.685} C_VEL
LIN {X 0,Y 531.135,Z 185.951,A -85,B 0,C 180,E1 -4497.725,E2 -4497.725} C_VEL
LIN {X 0,Y 531.15,Z 185.943,A -85,B 0,C 180,E1 -4500.758,E2 -4500.758} C_VEL
LIN {X 0,Y 531.103,Z 185.949,A -85,B 0,C 180,E1 -4503.034,E2 -4503.034} C_VEL
LIN {X 0,Y 531.081,Z 185.952,A -85,B 0,C 180,E1 -4506.077,E2 -4506.077} C_VEL
LIN {X 0,Y 531.028,Z 185.962,A -85,B 0,C 180,E1 -4509.138,E2 -4509.138} C_VEL
LIN {X 0,Y 531.038,Z 185.955,A -85,B 0,C 180,E1 -4512.225,E2 -4512.225} C_VEL
LIN {X 0,Y 530.993,Z 185.968,A -85,B 0,C 180,E1 -4515.35,E2 -4515.35} C_VEL
LIN {X 0,Y 530.987,Z 185.964,A -85,B 0,C 180,E1 -4518.521,E2 -4518.521} C_VEL
LIN {X 0,Y 530.998,Z 185.966,A -85,B 0,C 180,E1 -4520.938,E2 -4520.938} C_VEL
LIN {X 0,Y 530.97,Z 185.964,A -85,B 0,C 180,E1 -4524.225,E2 -4524.225} C_VEL
LIN {X 0,Y 531,Z 185.967,A -85,B 0,C 180,E1 -4526.744,E2 -4526.744} C_VEL
LIN {X 0,Y 530.98,Z 185.964,A -85,B 0,C 180,E1 -4529.323,E2 -4529.323} C_VEL
LIN {X 0,Y 530.964,Z 185.967,A -85,B 0,C 180,E1 -4532.101,E2 -4532.101} C_VEL
LIN {X 0,Y 530.988,Z 185.964,A -85,B 0,C 180,E1 -4534.854,E2 -4534.854} C_VEL
LIN {X 0,Y 530.966,Z 185.967,A -85,B 0,C 180,E1 -4537.508,E2 -4537.508} C_VEL
LIN {X 0,Y 530.98,Z 185.965,A -85,B 0,C 180,E1 -4540.433,E2 -4540.433} C_VEL
LIN {X 0,Y 530.96,Z 185.966,A -85,B 0,C 180,E1 -4543.281,E2 -4543.281} C_VEL
LIN {X 0,Y 530.951,Z 185.966,A -85,B 0,C 180,E1 -4543.567,E2 -4543.567} C_VEL
LIN {X 0,Y 530.281,Z 186.053,A -85,B 0,C 180,E1 -4544.2,E2 -4544.2} C_VEL
LIN {X 0,Y 527.436,Z 186.41,A -85,B 0,C 180,E1 -4545.229,E2 -4545.229} C_VEL
LIN {X 0,Y 525.034,Z 186.711,A -85,B 0,C 180,E1 -4546.058,E2 -4546.058} C_VEL
LIN {X 0,Y 524.002,Z 186.838,A -85,B 0,C 180,E1 -4546.697,E2 -4546.697} C_VEL
LIN {X 0,Y 523.917,Z 186.845,A -85,B 0,C 180,E1 -4546.914,E2 -4546.914} C_VEL
LIN {X 0,Y 523.949,Z 186.844,A -85,B 0,C 180,E1 -4549.921,E2 -4549.921} C_VEL
LIN {X 0,Y 523.909,Z 186.846,A -85,B 0,C 180,E1 -4552.868,E2 -4552.868} C_VEL
LIN {X 0,Y 523.941,Z 186.844,A -85,B 0,C 180,E1 -4555.711,E2 -4555.711} C_VEL
LIN {X 0,Y 523.922,Z 186.85,A -85,B 0,C 180,E1 -4558.456,E2 -4558.456} C_VEL
LIN {X 0,Y 523.928,Z 186.847,A -85,B 0,C 180,E1 -4561.125,E2 -4561.125} C_VEL
LIN {X 0,Y 523.986,Z 187.04,A -85,B 0,C 180,E1 -4563.246,E2 -4563.246} C_VEL
LIN {X 0,Y 526.65,Z 198.941,A -85,B 0,C 180,E1 -4565.155,E2 -4565.155} C_VEL
LIN {X 0,Y 526.022,Z 217.64,A -85,B 0,C 180,E1 -4567.825,E2 -4567.825} C_VEL
LIN {X 0,Y 525.367,Z 239.371,A -85,B 0,C 180,E1 -4570.868,E2 -4570.868} C_VEL
LIN {X 0,Y 525.296,Z 244.566,A -85,B 0,C 180,E1 -4571.554,E2 -4571.554} C_VEL
LIN {X 0,Y 527.449,Z 255.653,A -85,B 0,C 180,E1 -4571.805,E2 -4571.805} C_VEL
LIN {X 0,Y 526.9,Z 382.455,A -85,B 0,C 180,E1 -4573.534,E2 -4573.534} C_VEL
LIN {X 0,Y 526.647,Z 397.154,A -85,B 0,C 180,E1 -4573.884,E2 -4573.884} C_VEL
LIN {X 0,Y 526.412,Z 410.091,A -85,B 0,C 180,E1 -4574.345,E2 -4574.345} C_VEL
LIN {X 0,Y 526.105,Z 421.976,A -85,B 0,C 180,E1 -4574.901,E2 -4574.901} C_VEL
LIN {X 0,Y 525.61,Z 435.063,A -85,B 0,C 180,E1 -4575.678,E2 -4575.678} C_VEL
LIN {X 0,Y 525.209,Z 446.852,A -85,B 0,C 180,E1 -4576.556,E2 -4576.556} C_VEL
LIN {X 0,Y 524.844,Z 456.65,A -85,B 0,C 180,E1 -4577.432,E2 -4577.432} C_VEL
LIN {X 0,Y 524.465,Z 467.434,A -85,B 0,C 180,E1 -4578.6,E2 -4578.6} C_VEL
LIN {X 0,Y 524.105,Z 476.355,A -85,B 0,C 180,E1 -4579.765,E2 -4579.765} C_VEL
LIN {X 0,Y 523.836,Z 484.887,A -85,B 0,C 180,E1 -4581.124,E2 -4581.124} C_VEL
LIN {X 0,Y 523.686,Z 490.903,A -85,B 0,C 180,E1 -4582.287,E2 -4582.287} C_VEL
LIN {X 0,Y 523.545,Z 497.305,A -85,B 0,C 180,E1 -4583.835,E2 -4583.835} C_VEL
LIN {X 0,Y 523.395,Z 502.112,A -85,B 0,C 180,E1 -4585.379,E2 -4585.379} C_VEL
LIN {X 0,Y 523.419,Z 505.457,A -85,B 0,C 180,E1 -4586.921,E2 -4586.921} C_VEL
LIN {X 0,Y 523.273,Z 507.457,A -85,B 0,C 180,E1 -4588.46,E2 -4588.46} C_VEL
LIN {X 0,Y 523.257,Z 508.147,A -85,B 0,C 180,E1 -4590,E2 -4590} C_VEL
LIN {X 0,Y 523.271,Z 507.544,A -85,B 0,C 180,E1 -4591.539,E2 -4591.539} C_VEL
LIN {X 0,Y 523.418,Z 505.629,A -85,B 0,C 180,E1 -4593.078,E2 -4593.078} C_VEL
LIN {X 0,Y 523.394,Z 502.356,A -85,B 0,C 180,E1 -4594.621,E2 -4594.621} C_VEL
LIN {X 0,Y 523.54,Z 497.63,A -85,B 0,C 180,E1 -4596.165,E2 -4596.165} C_VEL
LIN {X 0,Y 523.606,Z 493.094,A -85,B 0,C 180,E1 -4597.325,E2 -4597.325} C_VEL
LIN {X 0,Y 523.788,Z 486.495,A -85,B 0,C 180,E1 -4598.681,E2 -4598.681} C_VEL
LIN {X 0,Y 524.047,Z 478.297,A -85,B 0,C 180,E1 -4600.04,E2 -4600.04} C_VEL
LIN {X 0,Y 524.362,Z 469.771,A -85,B 0,C 180,E1 -4601.206,E2 -4601.206} C_VEL
LIN {X 0,Y 524.733,Z 459.447,A -85,B 0,C 180,E1 -4602.374,E2 -4602.374} C_VEL
LIN {X 0,Y 525.164,Z 447.904,A -85,B 0,C 180,E1 -4603.445,E2 -4603.445} C_VEL
LIN {X 0,Y 525.578,Z 436.349,A -85,B 0,C 180,E1 -4604.322,E2 -4604.322} C_VEL
LIN {X 0,Y 525.979,Z 425.353,A -85,B 0,C 180,E1 -4605.003,E2 -4605.003} C_VEL
LIN {X 0,Y 526.344,Z 412.398,A -85,B 0,C 180,E1 -4605.645,E2 -4605.645} C_VEL
LIN {X 0,Y 526.635,Z 398.546,A -85,B 0,C 180,E1 -4606.16,E2 -4606.16} C_VEL
LIN {X 0,Y 526.879,Z 384.517,A -85,B 0,C 180,E1 -4606.516,E2 -4606.516} C_VEL
LIN {X 0,Y 527.087,Z 344.663,A -85,B 0,C 180,E1 -4607.082,E2 -4607.082} C_VEL
LIN {X 0,Y 527.386,Z 255.496,A -85,B 0,C 180,E1 -4608.289,E2 -4608.289} C_VEL
LIN {X 0,Y 525.326,Z 244.562,A -85,B 0,C 180,E1 -4608.535,E2 -4608.535} C_VEL
LIN {X 0,Y 525.82,Z 224.102,A -85,B 0,C 180,E1 -4611.359,E2 -4611.359} C_VEL
LIN {X 0,Y 526.55,Z 202.374,A -85,B 0,C 180,E1 -4614.441,E2 -4614.441} C_VEL
LIN {X 0,Y 526.583,Z 198.583,A -85,B 0,C 180,E1 -4614.992,E2 -4614.992} C_VEL
LIN {X 0,Y 523.949,Z 186.93,A -85,B 0,C 180,E1 -4616.89,E2 -4616.89} C_VEL
LIN {X 0,Y 523.94,Z 186.839,A -85,B 0,C 180,E1 -4619.755,E2 -4619.755} C_VEL
LIN {X 0,Y 523.932,Z 186.84,A -85,B 0,C 180,E1 -4622.449,E2 -4622.449} C_VEL
LIN {X 0,Y 523.931,Z 186.845,A -85,B 0,C 180,E1 -4625.225,E2 -4625.225} C_VEL
LIN {X 0,Y 523.913,Z 186.848,A -85,B 0,C 180,E1 -4628.101,E2 -4628.101} C_VEL
LIN {X 0,Y 523.939,Z 186.845,A -85,B 0,C 180,E1 -4631.091,E2 -4631.091} C_VEL
LIN {X 0,Y 523.935,Z 186.843,A -85,B 0,C 180,E1 -4634.227,E2 -4634.227} C_VEL
LIN {X 0,Y 523.913,Z 186.844,A -85,B 0,C 180,E1 -4636.832,E2 -4636.832} C_VEL
LIN {X 0,Y 523.94,Z 186.844,A -85,B 0,C 180,E1 -4638.908,E2 -4638.908} C_VEL
LIN {X 0,Y 523.912,Z 186.848,A -85,B 0,C 180,E1 -4641.898,E2 -4641.898} C_VEL
LIN {X 0,Y 523.934,Z 186.844,A -85,B 0,C 180,E1 -4644.908,E2 -4644.908} C_VEL
LIN {X 0,Y 523.932,Z 186.845,A -85,B 0,C 180,E1 -4647.679,E2 -4647.679} C_VEL
LIN {X 0,Y 523.964,Z 186.837,A -85,B 0,C 180,E1 -4650.673,E2 -4650.673} C_VEL
LIN {X 0,Y 523.969,Z 186.839,A -85,B 0,C 180,E1 -4653.728,E2 -4653.728} C_VEL
LIN {X 0,Y 523.93,Z 186.842,A -85,B 0,C 180,E1 -4656.27,E2 -4656.27} C_VEL
LIN {X 0,Y 523.94,Z 186.848,A -85,B 0,C 180,E1 -4658.766,E2 -4658.766} C_VEL
LIN {X 0,Y 523.947,Z 186.844,A -85,B 0,C 180,E1 -4661.22,E2 -4661.22} C_VEL
LIN {X 0,Y 523.934,Z 186.84,A -85,B 0,C 180,E1 -4663.639,E2 -4663.639} C_VEL
LIN {X 0,Y 523.934,Z 186.843,A -85,B 0,C 180,E1 -4666.028,E2 -4666.028} C_VEL
LIN {X 0,Y 524.005,Z 186.836,A -85,B 0,C 180,E1 -4668.394,E2 -4668.394} C_VEL
LIN {X 0,Y 523.998,Z 186.833,A -85,B 0,C 180,E1 -4671.516,E2 -4671.516} C_VEL
LIN {X 0,Y 524.077,Z 186.832,A -85,B 0,C 180,E1 -4674.613,E2 -4674.613} C_VEL
LIN {X 0,Y 524.105,Z 186.819,A -85,B 0,C 180,E1 -4677.694,E2 -4677.694} C_VEL
LIN {X 0,Y 524.117,Z 186.82,A -85,B 0,C 180,E1 -4680.768,E2 -4680.768} C_VEL
LIN {X 0,Y 524.067,Z 186.826,A -85,B 0,C 180,E1 -4683.075,E2 -4683.075} C_VEL
LIN {X 0,Y 524.04,Z 186.833,A -85,B 0,C 180,E1 -4686.159,E2 -4686.159} C_VEL
LIN {X 0,Y 523.993,Z 186.833,A -85,B 0,C 180,E1 -4689.262,E2 -4689.262} C_VEL
LIN {X 0,Y 523.995,Z 186.838,A -85,B 0,C 180,E1 -4691.74,E2 -4691.74} C_VEL
LIN {X 0,Y 523.985,Z 186.835,A -85,B 0,C 180,E1 -4695.052,E2 -4695.052} C_VEL
LIN {X 0,Y 523.957,Z 186.845,A -85,B 0,C 180,E1 -4697.969,E2 -4697.969} C_VEL
LIN {X 0,Y 523.964,Z 186.839,A -85,B 0,C 180,E1 -4700.41,E2 -4700.41} C_VEL
LIN {X 0,Y 523.909,Z 186.845,A -85,B 0,C 180,E1 -4702.894,E2 -4702.894} C_VEL
LIN {X 0,Y 523.948,Z 186.842,A -85,B 0,C 180,E1 -4705.419,E2 -4705.419} C_VEL
LIN {X 0,Y 523.96,Z 186.843,A -85,B 0,C 180,E1 -4707.999,E2 -4707.999} C_VEL
LIN {X 0,Y 523.937,Z 186.841,A -85,B 0,C 180,E1 -4710.855,E2 -4710.855} C_VEL
LIN {X 0,Y 523.955,Z 186.845,A -85,B 0,C 180,E1 -4713.735,E2 -4713.735} C_VEL
LIN {X 0,Y 523.913,Z 186.843,A -85,B 0,C 180,E1 -4716.404,E2 -4716.404} C_VEL
LIN {X 0,Y 523.916,Z 186.846,A -85,B 0,C 180,E1 -4719.085,E2 -4719.085} C_VEL
LIN {X 0,Y 523.945,Z 186.839,A -85,B 0,C 180,E1 -4722.12,E2 -4722.12} C_VEL
LIN {X 0,Y 523.936,Z 186.846,A -85,B 0,C 180,E1 -4725.311,E2 -4725.311} C_VEL
LIN {X 0,Y 523.95,Z 186.842,A -85,B 0,C 180,E1 -4728.69,E2 -4728.69} C_VEL
LIN {X 0,Y 523.91,Z 186.847,A -85,B 0,C 180,E1 -4731.899,E2 -4731.899} C_VEL
LIN {X 0,Y 523.919,Z 186.839,A -85,B 0,C 180,E1 -4734.912,E2 -4734.912} C_VEL
LIN {X 0,Y 523.93,Z 186.84,A -85,B 0,C 180,E1 -4737.681,E2 -4737.681} C_VEL
LIN {X 0,Y 523.948,Z 186.799,A -85,B 0,C 180,E1 -4740.678,E2 -4740.678} C_VEL
LIN {X 0,Y 523.957,Z 187.052,A -85,B 0,C 180,E1 -4741.701,E2 -4741.701} C_VEL
LIN {X 0,Y 527.543,Z 201.414,A -85,B 0,C 180,E1 -4743.634,E2 -4743.634} C_VEL
LIN {X 0,Y 526.681,Z 227.205,A -85,B 0,C 180,E1 -4746.608,E2 -4746.608} C_VEL
LIN {X 0,Y 526.129,Z 244.927,A -85,B 0,C 180,E1 -4748.606,E2 -4748.606} C_VEL
LIN {X 0,Y 528.262,Z 257.911,A -85,B 0,C 180,E1 -4748.902,E2 -4748.902} C_VEL
LIN {X 0,Y 527.185,Z 411.297,A -85,B 0,C 180,E1 -4751.089,E2 -4751.089} C_VEL
LIN {X 0,Y 526.909,Z 427.318,A -85,B 0,C 180,E1 -4751.482,E2 -4751.482} C_VEL
LIN {X 0,Y 526.565,Z 442.606,A -85,B 0,C 180,E1 -4752.023,E2 -4752.023} C_VEL
LIN {X 0,Y 526.16,Z 455.452,A -85,B 0,C 180,E1 -4752.611,E2 -4752.611} C_VEL
LIN {X 0,Y 525.762,Z 469.177,A -85,B 0,C 180,E1 -4753.398,E2 -4753.398} C_VEL
LIN {X 0,Y 525.32,Z 482.291,A -85,B 0,C 180,E1 -4754.32,E2 -4754.32} C_VEL
LIN {X 0,Y 524.887,Z 494.602,A -85,B 0,C 180,E1 -4755.362,E2 -4755.362} C_VEL
LIN {X 0,Y 524.509,Z 505.315,A -85,B 0,C 180,E1 -4756.439,E2 -4756.439} C_VEL
LIN {X 0,Y 524.18,Z 515.226,A -85,B 0,C 180,E1 -4757.613,E2 -4757.613} C_VEL
LIN {X 0,Y 523.942,Z 524.934,A -85,B 0,C 180,E1 -4758.981,E2 -4758.981} C_VEL
LIN {X 0,Y 523.688,Z 533.001,A -85,B 0,C 180,E1 -4760.343,E2 -4760.343} C_VEL
LIN {X 0,Y 523.547,Z 540.521,A -85,B 0,C 180,E1 -4761.898,E2 -4761.898} C_VEL
LIN {X 0,Y 523.468,Z 546.549,A -85,B 0,C 180,E1 -4763.47,E2 -4763.47} C_VEL
LIN {X 0,Y 523.442,Z 550.009,A -85,B 0,C 180,E1 -4764.607,E2 -4764.607} C_VEL
LIN {X 0,Y 523.401,Z 553.579,A -85,B 0,C 180,E1 -4766.151,E2 -4766.151} C_VEL
LIN {X 0,Y 523.332,Z 555.922,A -85,B 0,C 180,E1 -4767.691,E2 -4767.691} C_VEL
LIN {X 0,Y 523.248,Z 557.098,A -85,B 0,C 180,E1 -4769.231,E2 -4769.231} C_VEL
LIN {X 0,Y 523.248,Z 557.097,A -85,B 0,C 180,E1 -4770.77,E2 -4770.77} C_VEL
LIN {X 0,Y 523.332,Z 555.918,A -85,B 0,C 180,E1 -4772.309,E2 -4772.309} C_VEL
LIN {X 0,Y 523.401,Z 553.573,A -85,B 0,C 180,E1 -4773.85,E2 -4773.85} C_VEL
LIN {X 0,Y 523.442,Z 550.008,A -85,B 0,C 180,E1 -4775.393,E2 -4775.393} C_VEL
LIN {X 0,Y 523.49,Z 545.13,A -85,B 0,C 180,E1 -4776.94,E2 -4776.94} C_VEL
LIN {X 0,Y 523.581,Z 538.803,A -85,B 0,C 180,E1 -4778.491,E2 -4778.491} C_VEL
LIN {X 0,Y 523.775,Z 530.848,A -85,B 0,C 180,E1 -4780.046,E2 -4780.046} C_VEL
LIN {X 0,Y 523.969,Z 522.363,A -85,B 0,C 180,E1 -4781.411,E2 -4781.411} C_VEL
LIN {X 0,Y 524.286,Z 512.126,A -85,B 0,C 180,E1 -4782.778,E2 -4782.778} C_VEL
LIN {X 0,Y 524.61,Z 501.658,A -85,B 0,C 180,E1 -4783.954,E2 -4783.954} C_VEL
LIN {X 0,Y 525.037,Z 489.32,A -85,B 0,C 180,E1 -4785.112,E2 -4785.112} C_VEL
LIN {X 0,Y 525.487,Z 476.505,A -85,B 0,C 180,E1 -4786.112,E2 -4786.112} C_VEL
LIN {X 0,Y 525.944,Z 462.682,A -85,B 0,C 180,E1 -4786.996,E2 -4786.996} C_VEL
LIN {X 0,Y 526.396,Z 448.317,A -85,B 0,C 180,E1 -4787.733,E2 -4787.733} C_VEL
LIN {X 0,Y 526.722,Z 433.466,A -85,B 0,C 180,E1 -4788.324,E2 -4788.324} C_VEL
LIN {X 0,Y 527.075,Z 418.191,A -85,B 0,C 180,E1 -4788.764,E2 -4788.764} C_VEL
LIN {X 0,Y 527.285,Z 402.009,A -85,B 0,C 180,E1 -4789.061,E2 -4789.061} C_VEL
LIN {X 0,Y 528.292,Z 257.671,A -85,B 0,C 180,E1 -4791.101,E2 -4791.101} C_VEL
LIN {X 0,Y 526.149,Z 244.972,A -85,B 0,C 180,E1 -4791.392,E2 -4791.392} C_VEL
LIN {X 0,Y 526.812,Z 221.862,A -85,B 0,C 180,E1 -4794.009,E2 -4794.009} C_VEL
LIN {X 0,Y 527.545,Z 201.406,A -85,B 0,C 180,E1 -4796.366,E2 -4796.366} C_VEL
LIN {X 0,Y 523.959,Z 187.047,A -85,B 0,C 180,E1 -4798.299,E2 -4798.299} C_VEL
LIN {X 0,Y 523.933,Z 186.806,A -85,B 0,C 180,E1 -4800.853,E2 -4800.853} C_VEL
LIN {X 0,Y 523.928,Z 186.845,A -85,B 0,C 180,E1 -4803.729,E2 -4803.729} C_VEL
LIN {X 0,Y 523.901,Z 186.845,A -85,B 0,C 180,E1 -4806.401,E2 -4806.401} C_VEL
LIN {X 0,Y 523.911,Z 186.836,A -85,B 0,C 180,E1 -4809.085,E2 -4809.085} C_VEL
LIN {X 0,Y 523.949,Z 186.841,A -85,B 0,C 180,E1 -4812.119,E2 -4812.119} C_VEL
LIN {X 0,Y 523.94,Z 186.843,A -85,B 0,C 180,E1 -4815.31,E2 -4815.31} C_VEL
